(*%%%%%%%%%%%%%% Call Robots to Tool and Give Them, Task ID, Fixture ID and Model ID %%%%%%%%%%%%%%%%%*)
	(* Perform Call To Tool*)
	Tool_Call_ForLoadRobots1:= Enable_Motion AND (NOT Cell_In_Services OR NOT Load_Robots_Clear1)
						AND Start_Load_Robots1 AND NOT Start_Load_Robots2 AND NOT Start_Weld_Robots AND NOT Start_Seal_Robots AND NOT Start_Stud_Robots
						AND NOT Start_Unload_Robots1 AND NOT Start_Unload_Robots2 AND NOT Start_TurntableA AND NOT Start_TurntableB;
	Tool_Call_ForLoadRobots2:= Enable_Motion AND (NOT Cell_In_Services OR NOT Load_Robots_Clear2)
						AND NOT Start_Load_Robots1 AND Start_Load_Robots2 AND NOT Start_Weld_Robots AND NOT Start_Seal_Robots AND NOT Start_Stud_Robots
						AND NOT Start_Unload_Robots1 AND NOT Start_Unload_Robots2 AND NOT Start_TurntableA AND NOT Start_TurntableB;
	Tool_Call_ForSealRobots:=Enable_Motion AND (NOT Cell_In_Services OR NOT Seal_Robots_Clear)
						AND NOT Start_Load_Robots1 AND NOT Start_Load_Robots2 AND NOT Start_Weld_Robots AND Start_Seal_Robots AND NOT Start_Stud_Robots
						AND NOT Start_Unload_Robots1 AND NOT Start_Unload_Robots2 AND NOT Start_TurntableA AND NOT Start_TurntableB;
	Tool_Call_ForStudRobots:=Enable_Motion AND (NOT Cell_In_Services OR NOT Stud_Robots_Clear)
						AND NOT Start_Load_Robots1 AND NOT Start_Load_Robots2 AND NOT Start_Weld_Robots AND NOT Start_Seal_Robots AND Start_Stud_Robots
						AND NOT Start_Unload_Robots1 AND NOT Start_Unload_Robots2 AND NOT Start_TurntableA AND NOT Start_TurntableB;
	Tool_Call_ForSweepA:= Enable_Motion AND (NOT Cell_In_Services OR NOT TurntableA_Clear)
						AND NOT Start_Load_Robots1 AND NOT Start_Load_Robots2 AND NOT Start_Weld_Robots AND NOT Start_Seal_Robots AND NOT Start_Stud_Robots
						AND NOT Start_Unload_Robots1 AND NOT Start_Unload_Robots2 AND Start_TurntableA AND NOT Start_TurntableB;
	Tool_Call_ForSweepB:= Enable_Motion AND (NOT Cell_In_Services OR NOT TurntableB_Clear)
						AND NOT Start_Load_Robots1 AND NOT Start_Load_Robots2 AND NOT Start_Weld_Robots AND NOT Start_Seal_Robots AND NOT Start_Stud_Robots
						AND NOT Start_Unload_Robots1 AND NOT Start_Unload_Robots2 AND NOT Start_TurntableA AND Start_TurntableB;
	Tool_Call_ForWeldRobots:= Enable_Motion AND (NOT Cell_In_Services OR NOT Weld_Robots_Clear)
						AND NOT Start_Load_Robots1 AND NOT Start_Load_Robots2 AND Start_Weld_Robots AND NOT Start_Seal_Robots AND NOT Start_Stud_Robots
						AND NOT Start_Unload_Robots1 AND NOT Start_Unload_Robots2 AND NOT Start_TurntableA AND NOT Start_TurntableB;
	Tool_Call_ForUnloadRobots1:= Enable_Motion AND (NOT Cell_In_Services OR NOT Unload_Robots_Clear1)
						AND NOT Start_Load_Robots1 AND NOT Start_Load_Robots2 AND NOT Start_Weld_Robots AND NOT Start_Seal_Robots AND NOT Start_Stud_Robots
						AND Start_Unload_Robots1 AND NOT Start_Unload_Robots2 AND NOT Start_TurntableA AND NOT Start_TurntableB;
	Tool_Call_ForUnloadRobots2:= Enable_Motion AND (NOT Cell_In_Services OR NOT Unload_Robots_Clear2)
						AND NOT Start_Load_Robots1 AND NOT Start_Load_Robots2 AND NOT Start_Weld_Robots AND NOT Start_Seal_Robots AND NOT Start_Stud_Robots
						AND NOT Start_Unload_Robots1 AND Start_Unload_Robots2 AND NOT Start_TurntableA AND NOT Start_TurntableB;



	(*Allow Robots to Proceed Into Tool*)
	(*!!!!!This is the final OK to allow Robots Into the Tool Area, So it Better Be Ready!!!!!!!*)
	IF Enable_Motion
		THEN
			IF Load_Robots_Proceed1 AND Load_Robots_WorkingOK1 AND Load_Robots_Clear2 AND Seal_Robots_Clear AND Stud_Robots_Clear AND Turntable_Clear AND Weld_Robots_Clear AND Unload_Robots_Clear
				THEN Robots_Clear_ToProceed:=TRUE;
			ELSIF Load_Robots_Proceed2 AND Load_Robots_WorkingOK2 AND Load_Robots_Clear1 AND Seal_Robots_Clear AND Stud_Robots_Clear AND Turntable_Clear AND Weld_Robots_Clear AND Unload_Robots_Clear
				THEN Robots_Clear_ToProceed:=TRUE;
			ELSIF Seal_Robots_Proceed AND Seal_Robots_WorkingOK AND Load_Robots_Clear AND Stud_Robots_Clear AND Turntable_Clear AND Weld_Robots_Clear AND Unload_Robots_Clear
				THEN Robots_Clear_ToProceed:=TRUE;
			ELSIF Stud_Robots_Proceed AND Stud_Robots_WorkingOK AND Load_Robots_Clear AND Seal_Robots_Clear AND Turntable_Clear AND Weld_Robots_Clear AND Unload_Robots_Clear
				THEN Robots_Clear_ToProceed:=TRUE;
			ELSIF Weld_Robots_Proceed AND Weld_Robots_WorkingOK AND Load_Robots_Clear AND Seal_Robots_Clear AND Stud_Robots_Clear AND Turntable_Clear AND Unload_Robots_Clear
				THEN Robots_Clear_ToProceed:=TRUE;
			ELSIF Unload_Robots_Proceed1 AND Unload_Robots_WorkingOK1 AND Load_Robots_Clear AND Seal_Robots_Clear AND Stud_Robots_Clear AND Turntable_Clear AND Weld_Robots_Clear AND Unload_Robots_Clear2
				THEN Robots_Clear_ToProceed:=TRUE;
			ELSIF Unload_Robots_Proceed2 AND Unload_Robots_WorkingOK2 AND Load_Robots_Clear AND Seal_Robots_Clear AND Stud_Robots_Clear AND Turntable_Clear AND Weld_Robots_Clear AND Unload_Robots_Clear1
				THEN Robots_Clear_ToProceed:=TRUE;
			ELSE Robots_Clear_ToProceed:= FALSE;
			END_IF;
		ELSE Robots_Clear_ToProceed:= FALSE;
	END_IF;

(*+++++++++++++++++++++++++++++++++++++++++++++++ Task Complete Acks ++++++++++++++++++++++++++*)
	(*1st Load Complete Ack*)
	Load_Complete1_Ack:= Load_Robots_Complete1 AND Load_Complete1;

	(*2nd Load Complete Ack*)
	Load_Complete2_Ack:= Load_Robots_Complete2 AND Load_Complete2;

	(*Seal Complete Ack*)
	Seal_Complete_Ack:= Seal_Robots_Complete AND Sealing_Complete;

	(*Stud Complete Ack*)
	Stud_Complete_Ack:= Stud_Robots_Complete AND Stud_Complete;

	(*Sweep Complete ACK*)
	TurnA_Complete_Ack := TurntableA_Complete AND TurntableA_At_Robot;
	TurnB_Complete_Ack := TurntableB_Complete AND TurntableB_At_Robot;

	(*Weld Complete Ack*)
	Weld_Complete_Ack:= Weld_Robots_Complete AND Welding_Complete;

	(*Unload Complete Ack*)
	Unload_Complete1_Ack:= Unload_Robots_Complete1 AND Unload_Complete;

	(*Unload Complete Ack*)
	Unload_Complete2_Ack:= Unload_Robots_Complete2 AND Unload_Complete;















(*end*)
END_ACTION

ACTION Status_and_Faults:



(*^^^^^^^^^^^^^^^^^^^^^^^^^^^^^^^^^^^^^^ General Visualization ^^^^^^^^^^^^^^^^^^^^^^^^^^^^^^^^^^^^*)
	(*For Ready to Load Indicators*)
		(*Flash when tool should be loaded but load is not complete*)
		IF In_Auto AND Tool_At_Home AND NOT Welding_Complete AND All_Robots_Clear AND NOT All_Sensors_On.2
			THEN
				Ready_To_Load:= Pulse_500mS;
				(*Go solid when tool has been loaded properly*)
				(*Go solid when tool is ready to be unloaded*)
		ELSIF In_Auto AND All_Robots_Clear  AND ((Tool_At_Home AND NOT Welding_Complete AND All_Sensors_On.2 AND NOT Enable_Motion)
			OR (Tool_At_Unload.0 AND Welding_Complete AND (Sealing_Complete OR Sealer_Bypass) AND (Stud_Complete OR Stud_Bypass) AND TurntableA_At_Robot AND NOT All_Sensors_Off))
			THEN
				Ready_To_Load:= TRUE;
		ELSE
				Ready_To_Load:= FALSE;
		END_IF;
	(*For Red Stack Light Indicators*)
		Red_Lamp_Req:= PPFaults<>0 OR CLFaulted.0 OR CLFaulted.4 OR (NOT Sealer_Bypass AND MAIN.SL01.Disp1_Volume_NotOK AND (MAIN.R1.Task_ID_Ack=Seal_Fix01)) OR Load_Seq01.Faulted;


	(*Status Banners*)
		(*1 - Check Parts On Sub Check*)
		IF In_Auto AND NOT In_Manual AND NOT Cycle_Complete AND Tool_At_Load.4
			AND NOT Start_Load_Robots1 AND NOT Start_Load_Robots2 AND NOT Start_Seal_Robots AND NOT Start_Stud_Robots AND NOT Start_TurntableA
			AND NOT Start_TurntableB AND NOT Start_Weld_Robots AND NOT Start_Unload_Robots1 AND NOT Start_Unload_Robots2
			THEN
				IF NOT Dry_Cycle AND NOT All_Sensors_On.0
					THEN Status:= 1;
				ELSIF Dry_Cycle AND NOT Load_Complete1
					THEN Status:=1;
				END_IF;
		END_IF;
		(*2 - Sub Check OK*)
		IF In_Auto AND NOT In_Manual AND NOT Cycle_Complete AND Tool_At_Load.5
			AND NOT Start_Load_Robots1 AND NOT Start_Load_Robots2 AND NOT Start_Seal_Robots AND NOT Start_Stud_Robots AND NOT Start_TurntableA
			AND NOT Start_TurntableB AND NOT Start_Weld_Robots AND NOT Start_Unload_Robots1 AND NOT Start_Unload_Robots2
			THEN
				IF NOT Dry_Cycle AND NOT All_Sensors_On.1
					THEN Status:= 2;
				ELSIF Dry_Cycle AND NOT Load_Complete2
					THEN Status:=2;
				END_IF;
		END_IF;
		(*3 - Load Main Part*)
		IF In_Auto AND NOT In_Manual AND NOT Cycle_Complete AND Tool_At_Home
			AND NOT Start_Load_Robots1 AND NOT Start_Load_Robots2 AND NOT Start_Seal_Robots AND NOT Start_Stud_Robots AND NOT Start_TurntableA
			AND NOT Start_TurntableB AND NOT Start_Weld_Robots AND NOT Start_Unload_Robots1 AND NOT Start_Unload_Robots2
			THEN
				IF NOT Dry_Cycle AND NOT All_Sensors_On.2
					THEN Status:= 3;
				ELSIF Dry_Cycle AND NOT Load_Complete
					THEN Status:=3;
				END_IF;
		END_IF;
		(*10 - Load Parts Onto Tool*)
		IF In_Auto AND NOT In_Manual AND NOT Cycle_Complete AND Tool_At_Load.0
			AND NOT Start_Load_Robots1 AND NOT Start_Load_Robots2 AND NOT Start_Seal_Robots AND NOT Start_Stud_Robots AND NOT Start_TurntableA
			AND NOT Start_TurntableB AND NOT Start_Weld_Robots AND NOT Start_Unload_Robots1 AND NOT Start_Unload_Robots2
			THEN
				IF NOT Dry_Cycle AND NOT All_Sensors_On.2
					THEN Status:= 10;
				ELSIF Dry_Cycle AND NOT Load_Complete
					THEN Status:=10;
				END_IF;
		END_IF;
		(*11 - Robot(s) Loading*)
		IF ((Start_Load_Robots1 OR  Load_Robots_WorkingOK1) OR (Start_Load_Robots2 OR  Load_Robots_WorkingOK2)) AND In_Auto AND NOT In_Manual
			AND NOT Start_Seal_Robots AND NOT Start_Stud_Robots AND NOT Start_TurntableA
			AND NOT Start_TurntableB AND NOT Start_Weld_Robots AND NOT Start_Unload_Robots1 AND NOT Start_Unload_Robots2
			THEN Status:= 11;
		END_IF;
		(*12 - Parts Loaded OK*)
		IF In_Auto AND NOT In_Manual AND NOT Cycle_Complete
			AND NOT Start_Load_Robots1 AND NOT Start_Load_Robots2 AND NOT Start_Seal_Robots AND NOT Start_Stud_Robots AND NOT Start_TurntableA
			 AND NOT Start_TurntableB AND NOT Start_Weld_Robots AND NOT Start_Unload_Robots1 AND NOT Start_Unload_Robots2
			THEN
				IF (All_Sensors_On.2 AND Tool_At_Load.1) AND NOT Dry_Cycle
					THEN Status:= 12;
				ELSIF Load_Complete
					THEN Status:= 12;
				END_IF;
		END_IF;
		(*19 - Robot(s) Stud*)
		IF (Start_Stud_Robots OR Stud_Robots_WorkingOK) AND In_Auto AND NOT In_Manual
			AND NOT Start_Load_Robots1 AND NOT Start_Load_Robots2 AND NOT Start_Weld_Robots AND NOT Start_Seal_Robots AND NOT Start_TurntableA
			 AND NOT Start_TurntableB AND NOT Start_Unload_Robots1 AND NOT Start_Unload_Robots2
			THEN Status:= 19;
		END_IF;
		(*20 - Robot(s) Sealing*)
		IF (Start_Seal_Robots OR Seal_Robots_WorkingOK) AND In_Auto AND NOT In_Manual
			AND NOT Start_Load_Robots1 AND NOT Start_Load_Robots2 AND NOT Start_Weld_Robots AND NOT Start_Stud_Robots AND NOT Start_TurntableA
			 AND NOT Start_TurntableB AND NOT Start_Unload_Robots1 AND NOT Start_Unload_Robots2
			THEN Status:= 20;
		END_IF;
		(*21 - Robot(s) Welding*)
		IF (Start_Weld_Robots OR Weld_Robots_WorkingOK) AND In_Auto AND NOT In_Manual
			AND NOT Start_Load_Robots1 AND NOT Start_Load_Robots2 AND NOT Start_Seal_Robots AND NOT Start_Stud_Robots AND NOT Start_TurntableA
			 AND NOT Start_TurntableB AND NOT Start_Unload_Robots1 AND NOT Start_Unload_Robots2
			THEN Status:= 21;
		END_IF;
		(*22 - Welding Complete / Ready for Unload*)
		IF In_Auto AND NOT In_Manual AND NOT Cycle_Complete AND Welding_Complete AND (Sub1_Weld_Complete OR Sub2_Weld_Complete OR Sub3_Weld_Complete OR Sub4_Weld_Complete OR Sub5_Weld_Complete)
			AND NOT Start_Load_Robots1 AND NOT Start_Load_Robots2 AND NOT Start_Seal_Robots AND NOT Start_Stud_Robots AND NOT Start_TurntableA
			AND NOT Start_TurntableB AND NOT Start_Weld_Robots AND NOT Start_Unload_Robots1 AND NOT Start_Unload_Robots2 AND TurntableA_At_Robot
			THEN Status:= 22;
		END_IF;
		(*26 - Ready for Rotate*)
		IF (Start_TurntableA OR Start_TurntableB) AND In_Auto AND NOT In_Manual
			AND NOT Start_Load_Robots1 AND NOT Start_Load_Robots2 AND NOT Start_Seal_Robots AND NOT Start_Stud_Robots
			AND NOT Start_Weld_Robots AND NOT Start_Unload_Robots1 AND NOT Start_Unload_Robots2
			THEN Status := 26;
		END_IF;
		(*31 - Robot(s) Unloading*)
		IF (Start_Unload_Robots1 OR Unload_Robots_WorkingOK1 OR Start_Unload_Robots2 OR Unload_Robots_WorkingOK2) AND In_Auto AND NOT In_Manual
			AND NOT Start_Load_Robots1 AND NOT Start_Load_Robots2 AND NOT Start_Seal_Robots AND NOT Start_Stud_Robots AND NOT Start_TurntableA
			AND NOT Start_TurntableB AND NOT Start_Weld_Robots
			THEN Status:= 31;
		END_IF;
		(*32 - Unload Complete*)
		IF In_Auto AND NOT In_Manual AND NOT Cycle_Complete AND Unload_Complete AND All_Sensors_Off
			AND NOT Start_Load_Robots1 AND NOT Start_Load_Robots2 AND NOT Start_Seal_Robots AND NOT Start_Stud_Robots AND NOT Start_TurntableA
			AND NOT Start_TurntableB AND NOT Start_Weld_Robots AND NOT Start_Unload_Robots1 AND NOT Start_Unload_Robots2
			THEN Status:= 32;
		END_IF;
		(*42 - Cycle Complete*)
		IF In_Auto AND NOT In_Manual AND Cycle_Complete AND All_Sensors_Off
			THEN Status:= 42;
		END_IF;
		(*50 - In Manual*)
		IF In_Manual
			THEN Status:= 50;
		END_IF;
		(*51 - Clamp Fault*)
		IF (CLFaults1>0 OR CLFaults2>0 OR CLFaults3>0 OR CLFaults4>0) AND In_Auto AND NOT In_Manual
			THEN Status:= 51;
		END_IF;
		(*52 - Part Present Sensor Fault*)
		IF PPFaults>0 AND In_Auto AND NOT In_Manual
			THEN Status:= 52;
		END_IF;
		(*53 - Nut Checks Failed Call QA*)
		IF QAChecks_Failed AND In_Auto AND NOT In_Manual
			THEN Status:= 53;
		END_IF;
		(*54 - Sealer Failed Call QA*)
		IF NOT Sealer_Bypass AND (MAIN.SL01.Disp1_Volume_NotOK AND (MAIN.R1.Task_ID_Ack=Seal_Fix01)) AND In_Auto AND NOT In_Manual
			THEN Status:= 54;
		END_IF;
		(*55 - Load Sequence Fault Call QA*)
		IF Load_Seq01.Faulted AND In_Auto AND NOT In_Manual
			THEN Status:= 55;
		END_IF;



(*$$$$$$$$$$$$$$$$$$$$$$$$$$$$$$$$$$$$$$$$$$$$$$$$$$$ Faults $$$$$$$$$$$$$$$$$$$$$$$$$$$$$$$$$$$$$$$$$$$$$$$$$$$$$$$*)

	(*Clamp/Cylider Faults Group 1*)
		IF CLFaults1>0
			THEN CLFaulted.1:=TRUE;
		ELSE
			CLFaulted.1:=FALSE;
		END_IF;
	(*Clamp/Cylider Faults Group 2*)
		IF CLFaults2>0
			THEN CLFaulted.2:=TRUE;
		ELSE
			CLFaulted.2:=FALSE;
		END_IF;
	(*Clamp/Cylider Faults Group 3*)
		IF CLFaults3>0
			THEN CLFaulted.3:=TRUE;
		ELSE
			CLFaulted.3:=FALSE;
		END_IF;
	(*Clamp/Cylinder Faults Group 4 - Reserved Flag for QA Check Motion Faults*)
		IF CLFaults4>0
			THEN CLFaulted.4:=TRUE;
		ELSE
			CLFaulted.4:=FALSE;
		END_IF;
	(*Bit 0 is designated as ANY Clamp Group Faulted*)
	IF CLFaulted.1 OR CLFaulted.2 OR CLFaulted.3
		THEN CLFaulted.0:= TRUE;
	ELSE CLFaulted.0 := FALSE;
	END_IF;

	(*Part Present Sensor Faults*)
		IF (PPFaults>0) OR (PPFaults1>0) OR (PPFaults2>0)
			THEN PPFaulted.0:=TRUE;
		ELSE
			PPFaulted.0:=FALSE;
		END_IF;
























(*end*)
END_ACTION

ACTION Task_Fix_Model_IDs:


	(*Develop Task IDs - See Global Variable, "TaskID_Record"*)

	IF (Start_Load_Robots1 OR Start_Load_Robots2) AND Enable_Motion
		THEN Task_ID:= Dropoff_Fix01;
	ELSIF Start_Seal_Robots AND Enable_Motion
		THEN Task_ID:= Seal_Fix01;
	ELSIF Start_Stud_Robots AND Enable_Motion
		THEN Task_ID:= Stud_Fix01;
	ELSIF Start_Weld_Robots AND Enable_Motion
		THEN Task_ID:= Weld_Fix01;
	ELSIF Start_TurnTableA AND Enable_Motion
		THEN Task_ID:= Sweep_Fix01;
	ELSIF (Start_Unload_Robots1 OR Start_Unload_Robots2) AND Enable_Motion
		THEN Task_ID:= Pickup_Fix01;
	ELSE Task_ID:= 0;
	END_IF;

	(*Develop Fixture ID*)
	Fix_ID:= N00.ID;					(*In Future Map Beckhoff Dip Switch Data From IP67 Block to Here*)

	(*Develop Model ID*)
	(*If there is no model, but running fix01, we need to set model for table sweep - then blanks modelID after*)
	IF All_Sensors_Off AND Turntable_Bypassed AND TurntableB_At_Robot
		THEN
		Model_ID:= 1;
		ELSE
		Model_ID:= Discrete_In.ModelData;
	END_IF
END_ACTION

ACTION Tool_States:


(*+++++++++++THIS AREA IS CUSTOM PER INSTALLATION AND WILL HAVE TO BE MODIFIED PER +++++++++++++*)
(*+++++++++++THIS AREA IS CUSTOM PER INSTALLATION AND WILL HAVE TO BE MODIFIED PER +++++++++++++*)


(*
						 MODEL ID MAP
					 -------------------
				Model ID :  Part ID  :   Tooling ID
					1  	 : 	 504     :     42
					2	 :   524     :	   42
					3	 :   543     :	   47
					4	 :   526     :	   46
					5	 :   536     :	   45
					6	 :   550     :	   44
					7	 :   571     :	   43
	
*)
	

	(*Tooling Position at Home*)
				Tool_At_HOME:= (((Model_ID=3) OR (Model_ID=10)) AND Clamp1RETD AND Clamp2RETD AND Clamp3RETD AND Clamp4RETD
							AND Clamp5RETD AND Clamp6RETD AND Clamp7RETD AND Clamp8RETD
							AND Clamp9RETD AND Clamp10RETD AND Clamp11RETD AND Clamp12RETD
							AND Clamp13RETD AND Clamp14RETD AND Clamp15RETD AND Clamp16RETD
							AND Clamp17RETD AND Clamp18RETD AND Clamp19RETD AND Clamp20RETD
							AND Clamp21RETD AND Clamp22RETD AND Clamp23RETD AND Clamp24RETD
							AND Clamp25RETD AND Clamp26RETD AND Clamp27RETD AND Clamp28RETD
							AND Clamp29RETD AND Clamp30RETD AND Clamp31RETD AND Clamp32RETD
							AND Clamp33RETD AND Clamp34RETD AND Clamp35RETD AND Clamp36RETD
							AND Clamp37RETD AND Clamp38RETD AND Pin1ADVD AND Pin2ADVD AND Pin3RETD 
							AND Pin4ADVD AND Pin5ADVD AND Pin6RETD AND Pin7ADVD AND Pin8ADVD
							AND Slide1ADVD AND Slide2ADVD AND Slide3RETD AND Slide4ADVD AND Slide5RETD AND Slide6ADVD
							AND Slide7RETD AND Slide8ADVD AND Slide9RETD AND Slide10RETD AND Slide11ADVD AND Slide12RETD
							AND Slide13RETD AND Slide14ADVD AND Slide15ADVD)
							OR
								(((Model_ID<>3) AND (Model_ID<>10)) AND Clamp1RETD AND Clamp2RETD AND Clamp3RETD AND Clamp4RETD
							AND Clamp5RETD AND Clamp6RETD AND Clamp7RETD AND Clamp8RETD
							AND Clamp9RETD AND Clamp10RETD AND Clamp11RETD AND Clamp12RETD
							AND Clamp13RETD AND Clamp14RETD AND Clamp15RETD AND Clamp16RETD
							AND Clamp17RETD AND Clamp18RETD AND Clamp19RETD AND Clamp20RETD
							AND Clamp21RETD AND Clamp22RETD AND Clamp23RETD AND Clamp24RETD
							AND Clamp25RETD AND Clamp26RETD AND Clamp27RETD AND Clamp28RETD
							AND Clamp29RETD AND Clamp30RETD AND Clamp31RETD AND Clamp32RETD
							AND Clamp33RETD AND Clamp34RETD AND Clamp35RETD AND Clamp36RETD
							AND Clamp37RETD AND Clamp38RETD AND Pin1ADVD AND Pin2RETD AND Pin3RETD 
							AND Pin4ADVD AND Pin5RETD AND Pin6RETD AND Pin7RETD AND Pin8ADVD
							AND Slide1ADVD AND Slide2ADVD AND Slide3RETD AND Slide4ADVD AND Slide5RETD AND Slide6ADVD
							AND Slide7RETD AND Slide8ADVD AND Slide9RETD AND Slide10RETD AND Slide11ADVD AND Slide12RETD
							AND Slide13RETD AND Slide14ADVD AND Slide15ADVD);		

						
	(*Tooling Position for Operator Load*)
	IF ((Model_ID=3) OR (Model_ID=10)) THEN
		
				Tool_At_Load.0:= Clamp1RETD AND Clamp2RETD AND Clamp3RETD AND Clamp4RETD
							AND Clamp5RETD AND Clamp6RETD AND Clamp7RETD AND Clamp8RETD
							AND Clamp9RETD AND Clamp10RETD AND Clamp11RETD AND Clamp12RETD
							AND Clamp13RETD AND Clamp14RETD AND Clamp15RETD AND Clamp16RETD
							AND Clamp17RETD AND Clamp18RETD AND Clamp19RETD AND Clamp20RETD
							AND Clamp21RETD AND Clamp22RETD AND Clamp23RETD AND Clamp24RETD
							AND Clamp25RETD AND Clamp26RETD AND Clamp27RETD AND Clamp28RETD
							AND Clamp29RETD AND Clamp30RETD AND Clamp31RETD AND Clamp32RETD
							AND Clamp33RETD AND Clamp34RETD AND Clamp35RETD AND Clamp36RETD
							AND Clamp37RETD AND Clamp38RETD AND Pin1ADVD AND Pin2ADVD AND Pin3RETD 
							AND Pin4ADVD AND Pin5ADVD AND Pin6RETD AND Pin7ADVD AND Pin8ADVD
							AND Slide1ADVD AND Slide2ADVD AND Slide3RETD AND Slide4ADVD AND Slide5RETD AND Slide6ADVD
							AND Slide7RETD AND Slide8ADVD AND Slide9RETD AND Slide10RETD AND Slide11ADVD AND Slide12RETD
							AND Slide13RETD AND Slide14ADVD AND Slide15ADVD;
		ELSE
			
				Tool_At_Load.0:= Clamp1RETD AND Clamp2RETD AND Clamp3RETD AND Clamp4RETD
							AND Clamp5RETD AND Clamp6RETD AND Clamp7RETD AND Clamp8RETD
							AND Clamp9RETD AND Clamp10RETD AND Clamp11RETD AND Clamp12RETD
							AND Clamp13RETD AND Clamp14RETD AND Clamp15RETD AND Clamp16RETD
							AND Clamp17RETD AND Clamp18RETD AND Clamp19RETD AND Clamp20RETD
							AND Clamp21RETD AND Clamp22RETD AND Clamp23RETD AND Clamp24RETD
							AND Clamp25RETD AND Clamp26RETD AND Clamp27RETD AND Clamp28RETD
							AND Clamp29RETD AND Clamp30RETD AND Clamp31RETD AND Clamp32RETD
							AND Clamp33RETD AND Clamp34RETD AND Clamp35RETD AND Clamp36RETD
							AND Clamp37RETD AND Clamp38RETD AND Pin1ADVD AND Pin2RETD AND Pin3RETD 
							AND Pin4ADVD AND Pin5RETD AND Pin6RETD AND Pin7RETD AND Pin8ADVD
							AND Slide1ADVD AND Slide2ADVD AND Slide3RETD AND Slide4ADVD AND Slide5RETD AND Slide6ADVD
							AND Slide7RETD AND Slide8ADVD AND Slide9RETD AND Slide10RETD AND Slide11ADVD AND Slide12RETD
							AND Slide13RETD AND Slide14ADVD AND Slide15ADVD;
							
	END_IF		
	
	(*Tooling Position at Load Complete*)
	IF ((Model_ID =1) OR (Model_ID=8) OR (Model_ID =2) OR (Model_ID=9)) THEN
		
				Tool_At_Load.1:= (Clamp1ADVD AND Clamp2ADVD AND Clamp3ADVD AND Clamp4ADVD AND Clamp5ADVD
							AND Clamp6ADVD AND Clamp7ADVD AND Clamp8RETD AND Clamp9ADVD AND Clamp10RETD
							AND Clamp11ADVD AND Clamp12ADVD AND Clamp13ADVD AND Clamp14ADVD AND Clamp15ADVD
							AND Clamp16ADVD AND Clamp17ADVD AND Clamp18ADVD AND Clamp19ADVD AND Clamp20ADVD
							AND Clamp21ADVD AND Clamp22ADVD AND Clamp23RETD AND Clamp24RETD AND Clamp25RETD
							AND Clamp26ADVD AND Clamp27RETD AND Clamp28ADVD AND Clamp29ADVD AND Clamp30ADVD
							AND Clamp31RETD AND Clamp32ADVD AND Clamp33ADVD AND Clamp34ADVD AND Clamp35ADVD
							AND Clamp36ADVD AND Clamp37ADVD AND Clamp38ADVD AND Pin1ADVD AND Pin2RETD
							AND Pin3RETD AND Pin4ADVD AND Pin5RETD AND Pin6RETD AND Pin7RETD AND Pin8ADVD
							AND Slide1ADVD AND Slide2ADVD AND Slide3ADVD AND Slide4ADVD AND Slide5ADVD
							AND Slide6ADVD AND Slide7ADVD AND Slide8ADVD AND Slide9ADVD AND Slide10ADVD
							AND Slide11ADVD AND Slide12ADVD AND Slide13ADVD AND Slide14ADVD AND Slide15ADVD)
							OR (*After Hand Clamps*)
							(Clamp1RETD AND Clamp2RETD AND Clamp3RETD AND Clamp4RETD AND Clamp5RETD
							AND Clamp6ADVD AND Clamp7RETD AND Clamp8RETD AND Clamp9ADVD AND Clamp10RETD
							AND Clamp11RETD AND Clamp12RETD AND Clamp13RETD AND Clamp14RETD AND Clamp15RETD
							AND Clamp16RETD AND Clamp17RETD AND Clamp18RETD AND Clamp19RETD AND Clamp20RETD
							AND Clamp21ADVD AND Clamp22RETD AND Clamp23RETD AND Clamp24RETD AND Clamp25RETD
							AND Clamp26RETD AND Clamp27RETD AND Clamp28RETD AND Clamp29RETD AND Clamp30ADVD
							AND Clamp31RETD AND Clamp32RETD AND Clamp33RETD AND Clamp34RETD AND Clamp35RETD
							AND Clamp36ADVD AND Clamp37RETD AND Clamp38RETD AND Pin1ADVD AND Pin2RETD
							AND Pin3RETD AND Pin4ADVD AND Pin5RETD AND Pin6RETD AND Pin7RETD AND Pin8ADVD
							AND Slide1ADVD AND Slide2ADVD AND Slide3RETD AND Slide4ADVD AND Slide5RETD
							AND Slide6ADVD AND Slide7RETD AND Slide8ADVD AND Slide9RETD AND Slide10RETD
							AND Slide11ADVD AND Slide12RETD AND Slide13RETD AND Slide14ADVD AND Slide15ADVD);
							
		ELSIF ((Model_ID=3) OR (Model_ID=10)) THEN
			
				Tool_At_Load.1:= Clamp1ADVD AND Clamp2ADVD AND Clamp3ADVD AND Clamp4ADVD AND Clamp5ADVD
							AND Clamp6ADVD AND Clamp7RETD AND Clamp8ADVD AND Clamp9ADVD AND Clamp10ADVD
							AND Clamp11ADVD AND Clamp12ADVD AND Clamp13ADVD AND Clamp14ADVD AND Clamp15ADVD
							AND Clamp16ADVD AND Clamp17ADVD AND Clamp18ADVD AND Clamp19ADVD AND Clamp20ADVD
							AND Clamp21ADVD AND Clamp22RETD AND Clamp23RETD AND Clamp24ADVD AND Clamp25RETD
							AND Clamp26RETD AND Clamp27ADVD AND Clamp28ADVD AND Clamp29ADVD AND Clamp30ADVD
							AND Clamp31ADVD AND Clamp32ADVD AND Clamp33ADVD AND Clamp34ADVD AND Clamp35RETD
							AND Clamp36ADVD AND Clamp37ADVD AND Clamp38ADVD AND Pin1ADVD AND Pin2ADVD
							AND Pin3ADVD AND Pin4ADVD AND Pin5ADVD AND Pin6ADVD AND Pin7ADVD AND Pin8ADVD
							AND Slide1ADVD AND Slide2ADVD AND Slide3ADVD AND Slide4ADVD AND Slide5ADVD
							AND Slide6ADVD AND Slide7ADVD AND Slide8ADVD AND Slide9ADVD AND Slide10ADVD
							AND Slide11ADVD AND Slide12ADVD AND Slide13ADVD AND Slide14ADVD AND Slide15ADVD
							OR (*After Hand Clamps*)
							(Clamp1RETD AND Clamp2RETD AND Clamp3RETD AND Clamp4RETD AND Clamp5RETD
							AND Clamp6ADVD AND Clamp7RETD AND Clamp8ADVD AND Clamp9ADVD AND Clamp10ADVD
							AND Clamp11RETD AND Clamp12RETD AND Clamp13RETD AND Clamp14RETD AND Clamp15RETD
							AND Clamp16RETD AND Clamp17RETD AND Clamp18RETD AND Clamp19RETD AND Clamp20RETD
							AND Clamp21ADVD AND Clamp22RETD AND Clamp23RETD AND Clamp24ADVD AND Clamp25RETD
							AND Clamp26RETD AND Clamp27ADVD AND Clamp28RETD AND Clamp29RETD AND Clamp30ADVD
							AND Clamp31ADVD AND Clamp32RETD AND Clamp33RETD AND Clamp34RETD AND Clamp35RETD
							AND Clamp36ADVD AND Clamp37RETD AND Clamp38RETD AND Pin1ADVD AND Pin2ADVD
							AND Pin3RETD AND Pin4ADVD AND Pin5ADVD AND Pin6RETD AND Pin7ADVD AND Pin8ADVD
							AND Slide1ADVD AND Slide2ADVD AND Slide3RETD AND Slide4ADVD AND Slide5RETD
							AND Slide6ADVD AND Slide7RETD AND Slide8ADVD AND Slide9RETD AND Slide10RETD
							AND Slide11ADVD AND Slide12RETD AND Slide13RETD AND Slide14ADVD AND Slide15ADVD);
							
		ELSIF 			   (Model_ID=4) OR (Model_ID=5) OR (Model_ID=6) OR (Model_ID=7)
						OR (Model_ID=11) OR (Model_ID=12) OR (Model_ID=13) OR (Model_ID=14)
						OR (Model_ID=15) OR (Model_ID=16) OR (Model_ID=17) OR (Model_ID=18)
						OR (Model_ID=19) OR (Model_ID=20) OR (Model_ID=21) OR (Model_ID=22) THEN
			
				Tool_At_Load.1:= (Clamp1ADVD AND Clamp2ADVD AND Clamp3ADVD AND Clamp4ADVD AND Clamp5ADVD
							AND Clamp6ADVD AND Clamp7ADVD AND Clamp8RETD AND Clamp9ADVD AND Clamp10RETD
							AND Clamp11ADVD AND Clamp12ADVD AND Clamp13ADVD AND Clamp14ADVD AND Clamp15ADVD
							AND Clamp16ADVD AND Clamp17ADVD AND Clamp18ADVD AND Clamp19ADVD AND Clamp20ADVD
							AND Clamp21ADVD AND Clamp22RETD AND Clamp23ADVD AND Clamp24RETD AND Clamp25ADVD
							AND Clamp26RETD AND Clamp27RETD AND Clamp28ADVD AND Clamp29ADVD AND Clamp30ADVD
							AND Clamp31RETD AND Clamp32ADVD AND Clamp33ADVD AND Clamp34ADVD AND Clamp35ADVD
							AND Clamp36ADVD AND Clamp37ADVD AND Clamp38ADVD AND Pin1ADVD AND Pin2RETD
							AND Pin3RETD AND Pin4ADVD AND Pin5RETD AND Pin6RETD AND Pin7RETD AND Pin8ADVD
							AND Slide1ADVD AND Slide2ADVD AND Slide3ADVD AND Slide4ADVD AND Slide5ADVD
							AND Slide6ADVD AND Slide7ADVD AND Slide8ADVD AND Slide9ADVD AND Slide10ADVD
							AND Slide11ADVD AND Slide12ADVD AND Slide13ADVD AND Slide14ADVD AND Slide15ADVD)
							OR (*After Hand Clamps*)
							(Clamp1RETD AND Clamp2RETD AND Clamp3RETD AND Clamp4RETD AND Clamp5RETD
							AND Clamp6ADVD AND Clamp7RETD AND Clamp8RETD AND Clamp9ADVD AND Clamp10RETD
							AND Clamp11RETD AND Clamp12RETD AND Clamp13RETD AND Clamp14RETD AND Clamp15RETD
							AND Clamp16RETD AND Clamp17RETD AND Clamp18RETD AND Clamp19RETD AND Clamp20RETD
							AND Clamp21ADVD AND Clamp22RETD AND Clamp23RETD AND Clamp24RETD AND Clamp25RETD
							AND Clamp26RETD AND Clamp27RETD AND Clamp28RETD AND Clamp29RETD AND Clamp30ADVD
							AND Clamp31RETD AND Clamp32RETD AND Clamp33RETD AND Clamp34RETD AND Clamp35RETD
							AND Clamp36ADVD AND Clamp37RETD AND Clamp38RETD AND Pin1ADVD AND Pin2RETD
							AND Pin3RETD AND Pin4ADVD AND Pin5RETD AND Pin6RETD AND Pin7RETD AND Pin8ADVD
							AND Slide1ADVD AND Slide2ADVD AND Slide3RETD AND Slide4ADVD AND Slide5RETD
							AND Slide6ADVD AND Slide7RETD AND Slide8ADVD AND Slide9RETD AND Slide10ADVD
							AND Slide11ADVD AND Slide12RETD AND Slide13RETD AND Slide14ADVD AND Slide15ADVD);
							
	END_IF
	

(*Unused tool state - for reference BdB*)
	Tool_At_Load.2:= ((Model_ID=4) //526
							AND Clamp1ADVD AND Clamp2ADVD AND Clamp3ADVD AND Clamp4ADVD AND Clamp5ADVD
							AND Clamp6ADVD AND Clamp7ADVD AND Clamp8RETD AND Clamp9ADVD AND Clamp10RETD
							AND Clamp11ADVD AND Clamp12ADVD AND Clamp13ADVD AND Clamp14ADVD AND Clamp15ADVD
							AND Clamp16ADVD AND Clamp17ADVD AND Clamp18ADVD AND Clamp19ADVD AND Clamp20ADVD
							AND Clamp21ADVD AND Clamp22RETD AND Clamp23ADVD AND Clamp24RETD AND Clamp25ADVD
							AND Clamp26RETD AND Clamp27RETD AND Clamp28ADVD AND Clamp29ADVD AND Clamp30ADVD
							AND Clamp31RETD AND Clamp32ADVD AND Clamp33ADVD AND Clamp34ADVD AND Clamp35ADVD
							AND Clamp36ADVD AND Clamp37ADVD AND Clamp38ADVD AND Pin1ADVD AND Pin2RETD
							AND Pin3RETD AND Pin4ADVD AND Pin5RETD AND Pin6RETD AND Pin7RETD AND Pin8ADVD
							AND Slide1ADVD AND Slide2ADVD (*AND Slide3ADVD*, tooling issues*) AND Slide4ADVD AND Slide5ADVD
							AND Slide6ADVD AND Slide7RETD (*AND Slide7ADVD, wrong way around*) AND Slide8ADVD AND Slide9ADVD AND Slide10ADVD
							AND Slide11ADVD (*AND Slide12ADVD AND Slide13ADVD* tooling issues*) AND Slide14ADVD AND Slide15ADVD);
	Tool_At_Load.3:= FALSE;
	Tool_At_Load.4:= FALSE;


	Tool_At_Seal.0:= FALSE;
	Tool_At_Seal.1:= FALSE;
	Tool_At_Seal.2:= FALSE;
	Tool_At_Seal.3:= FALSE;
	Tool_At_Seal.4:= FALSE;


	Tool_At_Stud.0:= FALSE;
	Tool_At_Stud.1:= FALSE;
	Tool_At_Stud.2:= FALSE;
	Tool_At_Stud.3:= FALSE;
	Tool_At_Stud.4:= FALSE;


	IF ((Model_ID =1) OR (Model_ID=8) OR (Model_ID =2) OR (Model_ID=9)) THEN
		
				Tool_At_Rotate.0:= Clamp1ADVD AND Clamp2ADVD AND Clamp3ADVD AND Clamp4ADVD AND Clamp5ADVD
							AND Clamp6ADVD AND Clamp7ADVD AND Clamp8RETD AND Clamp9ADVD AND Clamp10RETD
							AND Clamp11ADVD AND Clamp12ADVD AND Clamp13ADVD AND Clamp14ADVD AND Clamp15ADVD
							AND Clamp16ADVD AND Clamp17ADVD AND Clamp18ADVD AND Clamp19ADVD AND Clamp20ADVD
							AND Clamp21ADVD AND Clamp22ADVD AND Clamp23RETD AND Clamp24RETD AND Clamp25RETD
							AND Clamp26ADVD AND Clamp27RETD AND Clamp28ADVD AND Clamp29ADVD AND Clamp30ADVD
							AND Clamp31RETD AND Clamp32ADVD AND Clamp33ADVD AND Clamp34ADVD AND Clamp35ADVD
							AND Clamp36ADVD AND Clamp37ADVD AND Clamp38ADVD AND Pin1ADVD AND Pin2RETD
							AND Pin3RETD AND Pin4ADVD AND Pin5RETD AND Pin6RETD AND Pin7RETD AND Pin8ADVD
							AND Slide1ADVD AND Slide2ADVD AND Slide3ADVD AND Slide4ADVD AND Slide5ADVD
							AND Slide6ADVD AND Slide7ADVD AND Slide8ADVD AND Slide9ADVD AND Slide10RETD
							AND Slide11ADVD AND Slide12ADVD AND Slide13ADVD AND Slide14ADVD AND Slide15ADVD;
							
		ELSIF ((Model_ID=3) OR (Model_ID=10)) THEN
			
				Tool_At_Rotate.0:= Clamp1ADVD AND Clamp2ADVD AND Clamp3ADVD AND Clamp4ADVD AND Clamp5ADVD
							AND Clamp6ADVD AND Clamp7RETD AND Clamp8ADVD AND Clamp9ADVD AND Clamp10ADVD
							AND Clamp11ADVD AND Clamp12ADVD AND Clamp13ADVD AND Clamp14ADVD AND Clamp15ADVD
							AND Clamp16ADVD AND Clamp17ADVD AND Clamp18ADVD AND Clamp19ADVD AND Clamp20ADVD
							AND Clamp21ADVD AND Clamp22RETD AND Clamp23RETD AND Clamp24ADVD AND Clamp25RETD
							AND Clamp26RETD AND Clamp27ADVD AND Clamp28ADVD AND Clamp29ADVD AND Clamp30ADVD
							AND Clamp31ADVD AND Clamp32ADVD AND Clamp33ADVD AND Clamp34ADVD AND Clamp35RETD
							AND Clamp36ADVD AND Clamp37ADVD AND Clamp38ADVD AND Pin1ADVD AND Pin2ADVD
							AND Pin3ADVD AND Pin4ADVD AND Pin5ADVD AND Pin6ADVD AND Pin7ADVD AND Pin8ADVD
							AND Slide1ADVD AND Slide2ADVD AND Slide3ADVD AND Slide4ADVD AND Slide5ADVD
							AND Slide6ADVD AND Slide7ADVD AND Slide8ADVD AND Slide9ADVD AND Slide10RETD
							AND Slide11ADVD AND Slide12ADVD AND Slide13ADVD AND Slide14ADVD AND Slide15ADVD;
							
		ELSIF 			   (Model_ID=4) OR (Model_ID=5) OR (Model_ID=6) OR (Model_ID=7)
						OR (Model_ID=11) OR (Model_ID=12) OR (Model_ID=13) OR (Model_ID=14)
						OR (Model_ID=15) OR (Model_ID=16) OR (Model_ID=17) OR (Model_ID=18)
						OR (Model_ID=19) OR (Model_ID=20) OR (Model_ID=21) OR (Model_ID=22) THEN
			
				Tool_At_Rotate.0:= Clamp1ADVD AND Clamp2ADVD AND Clamp3ADVD AND Clamp4ADVD AND Clamp5ADVD
							AND Clamp6ADVD AND Clamp7ADVD AND Clamp8RETD AND Clamp9ADVD AND Clamp10RETD
							AND Clamp11ADVD AND Clamp12ADVD AND Clamp13ADVD AND Clamp14ADVD AND Clamp15ADVD
							AND Clamp16ADVD AND Clamp17ADVD AND Clamp18ADVD AND Clamp19ADVD AND Clamp20ADVD
							AND Clamp21ADVD AND Clamp22RETD AND Clamp23ADVD AND Clamp24RETD AND Clamp25ADVD
							AND Clamp26RETD AND Clamp27RETD AND Clamp28ADVD AND Clamp29ADVD AND Clamp30ADVD
							AND Clamp31RETD AND Clamp32ADVD AND Clamp33ADVD AND Clamp34ADVD AND Clamp35ADVD
							AND Clamp36ADVD AND Clamp37ADVD AND Clamp38ADVD AND Pin1ADVD AND Pin2RETD
							AND Pin3RETD AND Pin4ADVD AND Pin5RETD AND Pin6RETD AND Pin7RETD AND Pin8ADVD
							AND Slide1ADVD AND Slide2ADVD AND Slide3ADVD AND Slide4ADVD AND Slide5ADVD
							AND Slide6ADVD AND Slide7ADVD AND Slide8ADVD AND Slide9ADVD AND Slide10ADVD
							AND Slide11ADVD AND Slide12ADVD AND Slide13ADVD AND Slide14ADVD AND Slide15ADVD;
	END_IF
				
	Tool_At_Rotate.1:= Clamp1RETD AND Clamp2RETD AND Clamp3RETD AND Clamp4RETD
							AND Clamp5RETD AND Clamp6RETD AND Clamp7RETD AND Clamp8RETD
							AND Clamp9RETD AND Clamp10RETD AND Clamp11RETD AND Clamp12RETD
							AND Clamp13RETD AND Clamp14RETD AND Clamp15RETD AND Clamp16RETD
							AND Clamp17RETD AND Clamp18RETD AND Clamp19RETD AND Clamp20RETD
							AND Clamp21RETD AND Clamp22RETD AND Clamp23RETD AND Clamp24RETD
							AND Clamp25RETD AND Clamp26RETD AND Clamp27RETD AND Clamp28RETD
							AND Clamp29RETD AND Clamp30RETD AND Clamp31RETD AND Clamp32RETD
							AND Clamp33RETD AND Clamp34RETD AND Clamp35RETD AND Clamp36RETD
							AND Clamp37RETD AND Clamp38RETD AND Pin1ADVD AND Pin2RETD AND Pin3RETD 
							AND Pin4ADVD AND Pin5RETD AND Pin6RETD AND Pin7RETD AND Pin8ADVD
							AND Slide1ADVD AND Slide2ADVD AND Slide3RETD AND Slide4ADVD AND Slide5RETD AND Slide6ADVD
							AND Slide7RETD AND Slide8ADVD AND Slide9RETD AND Slide10RETD AND Slide11ADVD AND Slide12RETD
							AND Slide13RETD AND Slide14ADVD AND Slide15ADVD;
	Tool_At_Rotate.2:= FALSE;
	Tool_At_Rotate.3:= FALSE;
	Tool_At_Rotate.4:= FALSE;


	IF ((Model_ID =1) OR (Model_ID=8) OR (Model_ID =2) OR (Model_ID=9)) THEN
		
				Tool_At_Weld.0:= Clamp1ADVD AND Clamp2ADVD AND Clamp3ADVD AND Clamp4ADVD AND Clamp5ADVD
							AND Clamp6ADVD AND Clamp7ADVD AND Clamp8RETD AND Clamp9ADVD AND Clamp10RETD
							AND Clamp11ADVD AND Clamp12ADVD AND Clamp13ADVD AND Clamp14ADVD AND Clamp15ADVD
							AND Clamp16ADVD AND Clamp17ADVD AND Clamp18ADVD AND Clamp19ADVD AND Clamp20ADVD
							AND Clamp21ADVD AND Clamp22ADVD AND Clamp23RETD AND Clamp24RETD AND Clamp25RETD
							AND Clamp26ADVD AND Clamp27RETD AND Clamp28ADVD AND Clamp29ADVD AND Clamp30ADVD
							AND Clamp31RETD AND Clamp32ADVD AND Clamp33ADVD AND Clamp34ADVD AND Clamp35ADVD
							AND Clamp36ADVD AND Clamp37ADVD AND Clamp38ADVD AND Pin1ADVD AND Pin2RETD
							AND Pin3RETD AND Pin4ADVD AND Pin5RETD AND Pin6RETD AND Pin7RETD AND Pin8ADVD
							AND Slide1ADVD AND Slide2ADVD AND Slide3ADVD AND Slide4ADVD AND Slide5ADVD
							AND Slide6ADVD AND Slide7ADVD AND Slide8ADVD AND Slide9ADVD AND Slide10RETD
							AND Slide11ADVD AND Slide12ADVD AND Slide13ADVD AND Slide14ADVD AND Slide15ADVD;
							
		ELSIF ((Model_ID=3) OR (Model_ID=10)) THEN
			
				Tool_At_Weld.0:= Clamp1ADVD AND Clamp2ADVD AND Clamp3ADVD AND Clamp4ADVD AND Clamp5ADVD
							AND Clamp6ADVD AND Clamp7RETD AND Clamp8ADVD AND Clamp9ADVD AND Clamp10ADVD
							AND Clamp11ADVD AND Clamp12ADVD AND Clamp13ADVD AND Clamp14ADVD AND Clamp15ADVD
							AND Clamp16ADVD AND Clamp17ADVD AND Clamp18ADVD AND Clamp19ADVD AND Clamp20ADVD
							AND Clamp21ADVD AND Clamp22RETD AND Clamp23RETD AND Clamp24ADVD AND Clamp25RETD
							AND Clamp26RETD AND Clamp27ADVD AND Clamp28ADVD AND Clamp29ADVD AND Clamp30ADVD
							AND Clamp31ADVD AND Clamp32ADVD AND Clamp33ADVD AND Clamp34ADVD AND Clamp35RETD
							AND Clamp36ADVD AND Clamp37ADVD AND Clamp38ADVD AND Pin1ADVD AND Pin2ADVD
							AND Pin3ADVD AND Pin4ADVD AND Pin5ADVD AND Pin6ADVD AND Pin7ADVD AND Pin8ADVD
							AND Slide1ADVD AND Slide2ADVD AND Slide3ADVD AND Slide4ADVD AND Slide5ADVD
							AND Slide6ADVD AND Slide7ADVD AND Slide8ADVD AND Slide9ADVD AND Slide10RETD
							AND Slide11ADVD AND Slide12ADVD AND Slide13ADVD AND Slide14ADVD AND Slide15ADVD;
							
		ELSIF 			   (Model_ID=4) OR (Model_ID=5) OR (Model_ID=6) OR (Model_ID=7)
						OR (Model_ID=11) OR (Model_ID=12) OR (Model_ID=13) OR (Model_ID=14)
						OR (Model_ID=15) OR (Model_ID=16) OR (Model_ID=17) OR (Model_ID=18)
						OR (Model_ID=19) OR (Model_ID=20) OR (Model_ID=21) OR (Model_ID=22) THEN
			
				Tool_At_Weld.0:= Clamp1ADVD AND Clamp2ADVD AND Clamp3ADVD AND Clamp4ADVD AND Clamp5ADVD
							AND Clamp6ADVD AND Clamp7ADVD AND Clamp8RETD AND Clamp9ADVD AND Clamp10RETD
							AND Clamp11ADVD AND Clamp12ADVD AND Clamp13ADVD AND Clamp14ADVD AND Clamp15ADVD
							AND Clamp16ADVD AND Clamp17ADVD AND Clamp18ADVD AND Clamp19ADVD AND Clamp20ADVD
							AND Clamp21ADVD AND Clamp22RETD AND Clamp23ADVD AND Clamp24RETD AND Clamp25ADVD
							AND Clamp26RETD AND Clamp27RETD AND Clamp28ADVD AND Clamp29ADVD AND Clamp30ADVD
							AND Clamp31RETD AND Clamp32ADVD AND Clamp33ADVD AND Clamp34ADVD AND Clamp35ADVD
							AND Clamp36ADVD AND Clamp37ADVD AND Clamp38ADVD AND Pin1ADVD AND Pin2RETD
							AND Pin3RETD AND Pin4ADVD AND Pin5RETD AND Pin6RETD AND Pin7RETD AND Pin8ADVD
							AND Slide1ADVD AND Slide2ADVD AND Slide3ADVD AND Slide4ADVD AND Slide5ADVD
							AND Slide6ADVD AND Slide7ADVD AND Slide8ADVD AND Slide9ADVD AND Slide10ADVD
							AND Slide11ADVD AND Slide12ADVD AND Slide13ADVD AND Slide14ADVD AND Slide15ADVD;
	END_IF
				
	Tool_At_Weld.1:= FALSE;
	Tool_At_Weld.2:= FALSE;
	Tool_At_Weld.3:= FALSE;
	Tool_At_Weld.4:= FALSE;


	IF ((Model_ID =1) OR (Model_ID=8) OR (Model_ID =2) OR (Model_ID=9)) THEN
		
				Tool_At_Unload.0:= Clamp1ADVD AND Clamp2ADVD AND Clamp3RETD AND Clamp4ADVD AND Clamp5RETD
							AND Clamp6RETD AND Clamp7ADVD AND Clamp8RETD AND Clamp9RETD AND Clamp10RETD
							AND Clamp11ADVD AND Clamp12RETD AND Clamp13ADVD AND Clamp14ADVD AND Clamp15ADVD
							AND Clamp16ADVD AND Clamp17ADVD AND Clamp18ADVD AND Clamp19ADVD AND Clamp20RETD
							AND Clamp21RETD AND Clamp22RETD AND Clamp23RETD AND Clamp24RETD AND Clamp25RETD
							AND Clamp26RETD AND Clamp27RETD AND Clamp28RETD AND Clamp29ADVD AND Clamp30RETD
							AND Clamp31RETD AND Clamp32ADVD AND Clamp33ADVD AND Clamp34RETD AND Clamp35ADVD
							AND Clamp36RETD AND Clamp37ADVD AND Clamp38RETD AND Pin1RETD AND Pin2RETD
							AND Pin3RETD AND Pin4RETD AND Pin5RETD AND Pin6RETD AND Pin7RETD AND Pin8RETD
							AND Slide1RETD AND Slide2RETD AND Slide3RETD AND Slide4ADVD AND Slide5RETD
							AND Slide6RETD AND Slide7ADVD AND Slide8ADVD AND Slide9RETD AND Slide10RETD
							AND Slide11ADVD AND Slide12RETD AND Slide13RETD AND Slide14RETD AND Slide15RETD;
							
		ELSIF ((Model_ID=3) OR (Model_ID=10)) THEN
			
				Tool_At_Unload.0:= Clamp1ADVD AND Clamp2ADVD AND Clamp3RETD AND Clamp4ADVD AND Clamp5RETD
							AND Clamp6RETD AND Clamp7RETD AND Clamp8ADVD AND Clamp9RETD AND Clamp10ADVD
							AND Clamp11ADVD AND Clamp12RETD AND Clamp13ADVD AND Clamp14ADVD AND Clamp15ADVD
							AND Clamp16ADVD AND Clamp17ADVD AND Clamp18ADVD AND Clamp19ADVD AND Clamp20RETD
							AND Clamp21RETD AND Clamp22RETD AND Clamp23RETD AND Clamp24ADVD AND Clamp25RETD
							AND Clamp26RETD AND Clamp27ADVD AND Clamp28RETD AND Clamp29ADVD AND Clamp30RETD
							AND Clamp31ADVD AND Clamp32ADVD AND Clamp33ADVD AND Clamp34RETD AND Clamp35RETD
							AND Clamp36RETD AND Clamp37ADVD AND Clamp38RETD AND Pin1RETD AND Pin2RETD
							AND Pin3RETD AND Pin4RETD AND Pin5RETD AND Pin6RETD AND Pin7RETD AND Pin8RETD
							AND Slide1RETD AND Slide2RETD AND Slide3RETD AND Slide4ADVD AND Slide5RETD
							AND Slide6RETD AND Slide7ADVD AND Slide8ADVD AND Slide9RETD AND Slide10RETD
							AND Slide11ADVD AND Slide12RETD AND Slide13RETD AND Slide14RETD AND Slide15RETD;
							
		ELSIF 			   (Model_ID=4) OR (Model_ID=5) OR (Model_ID=6) OR (Model_ID=7)
						OR (Model_ID=11) OR (Model_ID=12) OR (Model_ID=13) OR (Model_ID=14)
						OR (Model_ID=15) OR (Model_ID=16) OR (Model_ID=17) OR (Model_ID=18)
						OR (Model_ID=19) OR (Model_ID=20) OR (Model_ID=21) OR (Model_ID=22) THEN
			
				Tool_At_Unload.0:= Clamp1ADVD AND Clamp2ADVD AND Clamp3RETD AND Clamp4ADVD AND Clamp5RETD
							AND Clamp6RETD AND Clamp7ADVD AND Clamp8RETD AND Clamp9RETD AND Clamp10RETD
							AND Clamp11ADVD AND Clamp12RETD AND Clamp13ADVD AND Clamp14ADVD AND Clamp15ADVD
							AND Clamp16ADVD AND Clamp17ADVD AND Clamp18ADVD AND Clamp19ADVD AND Clamp20RETD
							AND Clamp21RETD AND Clamp22RETD AND Clamp23RETD AND Clamp24RETD AND Clamp25RETD
							AND Clamp26RETD AND Clamp27RETD AND Clamp28RETD AND Clamp29ADVD AND Clamp30RETD
							AND Clamp31RETD AND Clamp32ADVD AND Clamp33ADVD AND Clamp34RETD AND Clamp35ADVD
							AND Clamp36RETD AND Clamp37ADVD AND Clamp38RETD AND Pin1RETD AND Pin2RETD
							AND Pin3RETD AND Pin4RETD AND Pin5RETD AND Pin6RETD AND Pin7RETD AND Pin8RETD
							AND Slide1RETD AND Slide2RETD AND Slide3RETD AND Slide4ADVD AND Slide5RETD
							AND Slide6RETD AND Slide7ADVD AND Slide8ADVD AND Slide9RETD AND Slide10RETD
							AND Slide11ADVD AND Slide12RETD AND Slide13RETD AND Slide14RETD AND Slide15RETD;
	END_IF
	(*After Robot Repo 89*)			
	IF ((Model_ID =1) OR (Model_ID=8) OR (Model_ID =2) OR (Model_ID=9)) THEN
		
				Tool_At_Unload.1:= Clamp1ADVD AND Clamp2ADVD AND Clamp3RETD AND Clamp4RETD AND Clamp5RETD
							AND Clamp6RETD AND Clamp7RETD AND Clamp8RETD AND Clamp9RETD AND Clamp10RETD
							AND Clamp11RETD AND Clamp12RETD AND Clamp13ADVD AND Clamp14ADVD AND Clamp15ADVD
							AND Clamp16ADVD AND Clamp17ADVD AND Clamp18ADVD AND Clamp19ADVD AND Clamp20RETD
							AND Clamp21RETD AND Clamp22RETD AND Clamp23RETD AND Clamp24RETD AND Clamp25RETD
							AND Clamp26RETD AND Clamp27RETD AND Clamp28RETD AND Clamp29RETD AND Clamp30RETD
							AND Clamp31RETD AND Clamp32ADVD AND Clamp33RETD AND Clamp34RETD AND Clamp35RETD
							AND Clamp36RETD AND Clamp37ADVD AND Clamp38RETD AND Pin1RETD AND Pin2RETD
							AND Pin3RETD AND Pin4RETD AND Pin5RETD AND Pin6RETD AND Pin7RETD AND Pin8RETD
							AND Slide1RETD AND Slide2RETD AND Slide3RETD AND Slide4RETD AND Slide5RETD
							AND Slide6RETD AND Slide7ADVD AND Slide8RETD AND Slide9RETD AND Slide10RETD
							AND Slide11RETD AND Slide12RETD AND Slide13RETD AND Slide14RETD AND Slide15RETD;
							
		ELSIF ((Model_ID=3) OR (Model_ID=10)) THEN
			
				Tool_At_Unload.1:= Clamp1ADVD AND Clamp2ADVD AND Clamp3RETD AND Clamp4RETD AND Clamp5RETD
							AND Clamp6RETD AND Clamp7RETD AND Clamp8ADVD AND Clamp9RETD AND Clamp10ADVD
							AND Clamp11RETD AND Clamp12RETD AND Clamp13ADVD AND Clamp14ADVD AND Clamp15ADVD
							AND Clamp16ADVD AND Clamp17ADVD AND Clamp18ADVD AND Clamp19ADVD AND Clamp20RETD
							AND Clamp21RETD AND Clamp22RETD AND Clamp23RETD AND Clamp24ADVD AND Clamp25RETD
							AND Clamp26RETD AND Clamp27ADVD AND Clamp28RETD AND Clamp29RETD AND Clamp30RETD
							AND Clamp31ADVD AND Clamp32ADVD AND Clamp33RETD AND Clamp34RETD AND Clamp35RETD
							AND Clamp36RETD AND Clamp37ADVD AND Clamp38RETD AND Pin1RETD AND Pin2RETD
							AND Pin3RETD AND Pin4RETD AND Pin5RETD AND Pin6RETD AND Pin7RETD AND Pin8RETD
							AND Slide1RETD AND Slide2RETD AND Slide3RETD AND Slide4RETD AND Slide5RETD
							AND Slide6RETD AND Slide7ADVD AND Slide8RETD AND Slide9RETD AND Slide10RETD
							AND Slide11RETD AND Slide12RETD AND Slide13RETD AND Slide14RETD AND Slide15RETD;
							
		ELSIF 			   (Model_ID=4) OR (Model_ID=5) OR (Model_ID=6) OR (Model_ID=7)
						OR (Model_ID=11) OR (Model_ID=12) OR (Model_ID=13) OR (Model_ID=14)
						OR (Model_ID=15) OR (Model_ID=16) OR (Model_ID=17) OR (Model_ID=18)
						OR (Model_ID=19) OR (Model_ID=20) OR (Model_ID=21) OR (Model_ID=22) THEN
			
				Tool_At_Unload.1:= Clamp1ADVD AND Clamp2ADVD AND Clamp3RETD AND Clamp4RETD AND Clamp5RETD
							AND Clamp6RETD AND Clamp7RETD AND Clamp8RETD AND Clamp9RETD AND Clamp10RETD
							AND Clamp11RETD AND Clamp12RETD AND Clamp13ADVD AND Clamp14ADVD AND Clamp15ADVD
							AND Clamp16ADVD AND Clamp17ADVD AND Clamp18ADVD AND Clamp19ADVD AND Clamp20RETD
							AND Clamp21RETD AND Clamp22RETD AND Clamp23RETD AND Clamp24RETD AND Clamp25RETD
							AND Clamp26RETD AND Clamp27RETD AND Clamp28RETD AND Clamp29RETD AND Clamp30RETD
							AND Clamp31RETD AND Clamp32ADVD AND Clamp33RETD AND Clamp34RETD AND Clamp35RETD
							AND Clamp36RETD AND Clamp37ADVD AND Clamp38RETD AND Pin1RETD AND Pin2RETD
							AND Pin3RETD AND Pin4RETD AND Pin5RETD AND Pin6RETD AND Pin7RETD AND Pin8RETD
							AND Slide1RETD AND Slide2RETD AND Slide3RETD AND Slide4RETD AND Slide5RETD
							AND Slide6RETD AND Slide7ADVD AND Slide8RETD AND Slide9RETD AND Slide10RETD
							AND Slide11RETD AND Slide12RETD AND Slide13RETD AND Slide14RETD AND Slide15RETD;
	END_IF
	
	Tool_At_Unload.2:= FALSE;
	Tool_At_Unload.3:= FALSE;
	Tool_At_Unload.4:= FALSE;

(*end*)
END_ACTION

ACTION Tool_VBSeq_Repos:
(*+++++++++++THIS AREA IS CUSTOM PER INSTALLATION AND WILL HAVE TO BE MODIFIED PER +++++++++++++*)
(*+++++++++++THIS AREA IS CUSTOM PER INSTALLATION AND WILL HAVE TO BE MODIFIED PER +++++++++++++*)

(*!!!!!!!!!!!!!!!!!!!!!!!!!!!!!!!!!!!!!!!!!! Tool Motion Control !!!!!!!!!!!!!!!!!!!!!!!!!!!!!!!*)

(*----------------------------------------- Camp / Unclamp Steps -------------------------------*)

(*$$$$$$$$$$$$$$$$$$$$$$$$$$$$$$$$$$ Develop Clamp and Unclamp Interlocks $$$$$$$$$$$$$$$$$$$$$$*)
(* Note: This is one method to create valve bank commands for clamp and unclamp sequencing you are welcome to use the direct method as well*)

(*Start Clamp Sequence*)	
	
	(*First Stage Clamping*) (*V10, V11, V14, V15 ADV, IF Model 543, V19 ADV*)
		Clamp_Step.0:= Auto_Run AND (NOT Welding_Complete OR (Cycle_Complete AND NOT Tool_At_Home)) AND NOT All_Sensors_Off;

	(*Second Stage Clamping*)	(*V12, V13 ADV, IF Model 543, V20, V21 ADV*)
		(*504*)
			IF ((Model_ID=1) OR (Model_ID=8)) THEN
						Clamp_Step.1:=  Clamp_Step.0 AND 
										(*V10*)
										(Slide4ADVD AND Slide8ADVD AND Slide11ADVD)
										(*V11*)
										AND (Slide6ADVD)
										(*V14*)
										AND (Slide1ADVD AND Slide2ADVD AND Slide14ADVD AND Slide15ADVD)
										(*V15*)
										AND (Pin1ADVD AND Pin4ADVD AND Pin8ADVD);
		(*524*)						
				ELSIF ((Model_ID=2) OR (Model_ID=9)) THEN
						Clamp_Step.1:=  Clamp_Step.0 AND 
										(*V10*)
										(Slide4ADVD AND Slide8ADVD AND Slide11ADVD)
										(*V11*)
										AND (Slide6ADVD)
										(*V14*)
										AND (Slide1ADVD AND Slide2ADVD AND Slide14ADVD AND Slide15ADVD)
										(*V15*)
										AND (Pin1ADVD AND Pin4ADVD AND Pin8ADVD);
		(*543*)						
				ELSIF ((Model_ID=3) OR (Model_ID=10)) THEN
						Clamp_Step.1:=  Clamp_Step.0 AND 
										(*V10*)
										(Slide4ADVD AND Slide8ADVD AND Slide11ADVD)
										(*V11*)
										AND (Slide6ADVD)
										(*V14*)
										AND (Slide1ADVD AND Slide2ADVD AND Slide14ADVD AND Slide15ADVD)
										(*V15*)
										AND (Pin1ADVD AND Pin4ADVD AND Pin8ADVD)
										(*V19*)
										AND (Pin2ADVD AND Pin5ADVD AND Pin7ADVD);
		(*526*)						
				ELSIF ((Model_ID=4) OR (Model_ID=11) OR (Model_ID=15) OR (Model_ID=19)) THEN
						Clamp_Step.1:=  Clamp_Step.0 AND 
										(*V10*)
										(Slide4ADVD AND Slide8ADVD AND Slide11ADVD)
										(*V11*)
										AND (Slide6ADVD)
										(*V14*)
										AND (Slide1ADVD AND Slide2ADVD AND Slide14ADVD AND Slide15ADVD)
										(*V15*)
										AND (Pin1ADVD AND Pin4ADVD AND Pin8ADVD);
		(*536*)						
				ELSIF ((Model_ID=5) OR (Model_ID=12) OR (Model_ID=16) OR (Model_ID=20)) THEN
						Clamp_Step.1:=  Clamp_Step.0 AND 
										(*V10*)
										(Slide4ADVD AND Slide8ADVD AND Slide11ADVD)
										(*V11*)
										AND (Slide6ADVD)
										(*V14*)
										AND (Slide1ADVD AND Slide2ADVD AND Slide14ADVD AND Slide15ADVD)
										(*V15*)
										AND (Pin1ADVD AND Pin4ADVD AND Pin8ADVD);
		(*550*)						
				ELSIF ((Model_ID=6) OR (Model_ID=13) OR (Model_ID=17) OR (Model_ID=21)) THEN
						Clamp_Step.1:=  Clamp_Step.0 AND 
										(*V10*)
										(Slide4ADVD AND Slide8ADVD AND Slide11ADVD)
										(*V11*)
										AND (Slide6ADVD)
										(*V14*)
										AND (Slide1ADVD AND Slide2ADVD AND Slide14ADVD AND Slide15ADVD)
										(*V15*)
										AND (Pin1ADVD AND Pin4ADVD AND Pin8ADVD);
		(*571*)						
				ELSIF ((Model_ID=7) OR (Model_ID=14) OR (Model_ID=18) OR (Model_ID=22)) THEN
						Clamp_Step.1:=  Clamp_Step.0 AND 
										(*V10*)
										(Slide4ADVD AND Slide8ADVD AND Slide11ADVD)
										(*V11*)
										AND (Slide6ADVD)
										(*V14*)
										AND (Slide1ADVD AND Slide2ADVD AND Slide14ADVD AND Slide15ADVD)
										(*V15*)
										AND (Pin1ADVD AND Pin4ADVD AND Pin8ADVD);
			END_IF

	(*Third Stage Clamping*)	(*V1-V7 ADV, IF Model 504, 524, V8 ADV, IF Model 526, 536, 550, 571, V9 ADV, IF Model 543, V18 ADV*)
		(*504*)
			IF ((Model_ID=1) OR (Model_ID=8)) THEN
						Clamp_Step.2:= Clamp_Step.1 AND 
										(*V12*)
										(Slide7ADVD)
										(*V13*)
										AND (Slide10ADVD);
		(*524*)						
				ELSIF ((Model_ID=2) OR (Model_ID=9)) THEN
						Clamp_Step.2:= Clamp_Step.1 AND 
										(*V12*)
										(Slide7RETD)
										(*V13*)
										AND (Slide10ADVD);
		(*543*)				
				ELSIF ((Model_ID=3) OR (Model_ID=10)) THEN
						Clamp_Step.2:= Clamp_Step.1 AND 
										(*V12*)
										(Slide7ADVD)
										(*V13*)
										AND (Slide10ADVD)
										(*V20*)
										AND (Clamp8ADVD AND Clamp24ADVD AND Clamp31ADVD)
										(*V21*)
										AND (Clamp10ADVD AND Clamp27ADVD);
		(*526*)
				ELSIF ((Model_ID=4) OR (Model_ID=11) OR (Model_ID=15) OR (Model_ID=19)) THEN
						Clamp_Step.2:= Clamp_Step.1 AND 
										(*V12*)
										(Slide7RETD)
										(*V13*)
										AND (Slide10ADVD);
		(*536*)						
				ELSIF ((Model_ID=5) OR (Model_ID=12) OR (Model_ID=16) OR (Model_ID=20)) THEN
						Clamp_Step.2:= Clamp_Step.1 AND 
										(*V12*)
										(Slide7RETD)
										(*V13*)
										AND (Slide10ADVD);
		(*550*)						
				ELSIF ((Model_ID=6) OR (Model_ID=13) OR (Model_ID=17) OR (Model_ID=21)) THEN
						Clamp_Step.2:= Clamp_Step.1 AND 
										(*V12*)
										(Slide7RETD)
										(*V13*)
										AND (Slide10ADVD);
		(*571*)						
				ELSIF ((Model_ID=7) OR (Model_ID=14) OR (Model_ID=18) OR (Model_ID=22)) THEN
						Clamp_Step.2:= Clamp_Step.1 AND 
										(*V12*)
										(Slide7RETD)
										(*V13*)
										AND (Slide10ADVD);
			END_IF
														
	(*Forth Stage Clamping*)	(*Fire QAs - V17*)
		(*504*)	
			IF ((Model_ID=1) OR (Model_ID=8)) THEN
						Clamp_Step.3:= Clamp_Step.2 AND 
										(*V1*)
										(Clamp1ADVD AND Clamp2ADVD AND Clamp32ADVD AND Clamp37ADVD)
										(*V2*)
										AND (Clamp13ADVD AND Clamp14ADVD AND Clamp15ADVD)
										(*V3*)
										AND (Clamp16ADVD AND Clamp17ADVD AND Clamp18ADVD AND Clamp19ADVD)
										(*V4*)
										AND (Clamp3ADVD AND Clamp12ADVD AND Clamp20ADVD AND Clamp28ADVD AND Clamp34ADVD)
										(*V5*)
										AND (Clamp4ADVD AND Clamp11ADVD AND Clamp21ADVD AND Clamp29ADVD AND Clamp33ADVD)
										(*V6*)
										AND (Clamp6ADVD AND Clamp9ADVD AND Clamp30ADVD AND Clamp36ADVD)
										(*V7*)
										AND (Clamp7ADVD AND Clamp35ADVD)
										(*V8*)
										AND (Clamp22ADVD AND Clamp26ADVD);
		(*524*)						
				ELSIF ((Model_ID=2) OR (Model_ID=9)) THEN
						Clamp_Step.3:= Clamp_Step.2 AND 
										(*V1*)
										(Clamp1ADVD AND Clamp2ADVD AND Clamp32ADVD AND Clamp37ADVD)
										(*V2*)
										AND (Clamp13ADVD AND Clamp14ADVD AND Clamp15ADVD)
										(*V3*)
										AND (Clamp16ADVD AND Clamp17ADVD AND Clamp18ADVD AND Clamp19ADVD)
										(*V4*)
										AND (Clamp3ADVD AND Clamp12ADVD AND Clamp20ADVD AND Clamp28ADVD AND Clamp34ADVD)
										(*V5*)
										AND (Clamp4ADVD AND Clamp11ADVD AND Clamp21ADVD AND Clamp29ADVD AND Clamp33ADVD)
										(*V6*)
										AND (Clamp6ADVD AND Clamp9ADVD AND Clamp30ADVD AND Clamp36ADVD)
										(*V7*)
										AND (Clamp7ADVD AND Clamp35ADVD)
										(*V8*)
										AND (Clamp22ADVD AND Clamp26ADVD);								
		(*543*)						
				ELSIF ((Model_ID=3) OR (Model_ID=10)) THEN
						Clamp_Step.3:= Clamp_Step.2 AND 
										(*V1*)
										(Clamp1ADVD AND Clamp2ADVD AND Clamp32ADVD AND Clamp37ADVD)
										(*V2*)
										AND (Clamp13ADVD AND Clamp14ADVD AND Clamp15ADVD)
										(*V3*)
										AND (Clamp16ADVD AND Clamp17ADVD AND Clamp18ADVD AND Clamp19ADVD)
										(*V4*)
										AND (Clamp3ADVD AND Clamp12ADVD AND Clamp20ADVD AND Clamp28ADVD AND Clamp34ADVD)
										(*V5*)
										AND (Clamp4ADVD AND Clamp11ADVD AND Clamp21ADVD AND Clamp29ADVD AND Clamp33ADVD)
										(*V6*)
										AND (Clamp6ADVD AND Clamp9ADVD AND Clamp30ADVD AND Clamp36ADVD)
										(*V7*)
										AND (Clamp7ADVD AND Clamp35ADVD)
										(*V18*)
										AND (Pin3ADVD AND Pin6ADVD);
		(*526*)						
				ELSIF ((Model_ID=4) OR (Model_ID=11) OR (Model_ID=15) OR (Model_ID=19)) THEN
						Clamp_Step.3:= Clamp_Step.2 AND 
										(*V1*)
										(Clamp1ADVD AND Clamp2ADVD AND Clamp32ADVD AND Clamp37ADVD)
										(*V2*)
										AND (Clamp13ADVD AND Clamp14ADVD AND Clamp15ADVD)
										(*V3*)
										AND (Clamp16ADVD AND Clamp17ADVD AND Clamp18ADVD AND Clamp19ADVD)
										(*V4*)
										AND (Clamp3ADVD AND Clamp12ADVD AND Clamp20ADVD AND Clamp28ADVD AND Clamp34ADVD)
										(*V5*)
										AND (Clamp4ADVD AND Clamp11ADVD AND Clamp21ADVD AND Clamp29ADVD AND Clamp33ADVD)
										(*V6*)
										AND (Clamp6ADVD AND Clamp9ADVD AND Clamp30ADVD AND Clamp36ADVD)
										(*V7*)
										AND (Clamp7ADVD AND Clamp35ADVD)
										(*V9*)
										AND (Clamp23ADVD AND Clamp25ADVD);
		(*536*)						
				ELSIF ((Model_ID=5) OR (Model_ID=12) OR (Model_ID=16) OR (Model_ID=20)) THEN
						Clamp_Step.3:= Clamp_Step.2 AND 
										(*V1*)
										(Clamp1ADVD AND Clamp2ADVD AND Clamp32ADVD AND Clamp37ADVD)
										(*V2*)
										AND (Clamp13ADVD AND Clamp14ADVD AND Clamp15ADVD)
										(*V3*)
										AND (Clamp16ADVD AND Clamp17ADVD AND Clamp18ADVD AND Clamp19ADVD)
										(*V4*)
										AND (Clamp3ADVD AND Clamp12ADVD AND Clamp20ADVD AND Clamp28ADVD AND Clamp34ADVD)
										(*V5*)
										AND (Clamp4ADVD AND Clamp11ADVD AND Clamp21ADVD AND Clamp29ADVD AND Clamp33ADVD)
										(*V6*)
										AND (Clamp6ADVD AND Clamp9ADVD AND Clamp30ADVD AND Clamp36ADVD)
										(*V7*)
										AND (Clamp7ADVD AND Clamp35ADVD)
										(*V9*)
										AND (Clamp23ADVD AND Clamp25ADVD);
		(*550*)
				ELSIF ((Model_ID=6) OR (Model_ID=13) OR (Model_ID=17) OR (Model_ID=21)) THEN
						Clamp_Step.3:= Clamp_Step.2 AND 
										(*V1*)
										(Clamp1ADVD AND Clamp2ADVD AND Clamp32ADVD AND Clamp37ADVD)
										(*V2*)
										AND (Clamp13ADVD AND Clamp14ADVD AND Clamp15ADVD)
										(*V3*)
										AND (Clamp16ADVD AND Clamp17ADVD AND Clamp18ADVD AND Clamp19ADVD)
										(*V4*)
										AND (Clamp3ADVD AND Clamp12ADVD AND Clamp20ADVD AND Clamp28ADVD AND Clamp34ADVD)
										(*V5*)
										AND (Clamp4ADVD AND Clamp11ADVD AND Clamp21ADVD AND Clamp29ADVD AND Clamp33ADVD)
										(*V6*)
										AND (Clamp6ADVD AND Clamp9ADVD AND Clamp30ADVD AND Clamp36ADVD)
										(*V7*)
										AND (Clamp7ADVD AND Clamp35ADVD)
										(*V9*)
										AND (Clamp23ADVD AND Clamp25ADVD);
		(*571*)
				ELSIF ((Model_ID=7) OR (Model_ID=14) OR (Model_ID=18) OR (Model_ID=22)) THEN
						Clamp_Step.3:= Clamp_Step.2 AND 
										(*V1*)
										(Clamp1ADVD AND Clamp2ADVD AND Clamp32ADVD AND Clamp37ADVD)
										(*V2*)
										AND (Clamp13ADVD AND Clamp14ADVD AND Clamp15ADVD)
										(*V3*)
										AND (Clamp16ADVD AND Clamp17ADVD AND Clamp18ADVD AND Clamp19ADVD)
										(*V4*)
										AND (Clamp3ADVD AND Clamp12ADVD AND Clamp20ADVD AND Clamp28ADVD AND Clamp34ADVD)
										(*V5*)
										AND (Clamp4ADVD AND Clamp11ADVD AND Clamp21ADVD AND Clamp29ADVD AND Clamp33ADVD)
										(*V6*)
										AND (Clamp6ADVD AND Clamp9ADVD AND Clamp30ADVD AND Clamp36ADVD)
										(*V7*)
										AND (Clamp7ADVD AND Clamp35ADVD)
										(*V9*)
										AND (Clamp23ADVD AND Clamp25ADVD);								
			END_IF
	
	
	(*Fifth Stage Clamping*)	(*V16 ADV*)
			(*QA Check All Models*)
				Clamp_Step.4:= Clamp_Step.3 (*AND
					CheckQA1FB.QAcheck_OK*); (*Positions are off currently - AB*)
	
	
(*Start Unclamp Sequence*)
	(*First Stage Unclamping*)	(*V11, V13, V15, V16 RET, IF Model 543, V18, V19 RET*)
		Unclamp_Step.0:= (Welding_Complete AND TurnTableB_At_Robot AND NOT (MAIN.R1.Task_ID_Ack=Sweep_Fix01) AND NOT (MAIN.R1.Task_ID_Ack=Sweep_Fix03) AND NOT Cycle_Complete);
	
	(*Second Stage Unclamping*)	(*V4, V6, V14 RET, IF Model 504, 524, V8 RET, IF Model 526, 536, 550, 571, V9 RET*)
		(*504*)
			IF ((Model_ID=1) OR (Model_ID=8)) THEN
							Unclamp_Step.1:= Unclamp_Step.0 AND 
											(*V11*)
											(Slide6RETD)
											(*V13*)
											AND (Slide10RETD)
											(*V15*)
											AND (Pin1RETD AND Pin4RETD AND Pin8RETD)
											(*V16*)
											AND (Clamp5RETD AND Clamp38RETD AND Slide3RETD AND Slide5RETD AND Slide9RETD AND Slide12RETD AND Slide13RETD);
		(*524*)								
				ELSIF ((Model_ID=2) OR (Model_ID=9)) THEN
							Unclamp_Step.1:= Unclamp_Step.0 AND 
											(*V11*)
											(Slide6RETD)
											(*V13*)
											AND (Slide10RETD)
											(*V15*)
											AND (Pin1RETD AND Pin4RETD AND Pin8RETD)
											(*V16*)
											AND (Clamp5RETD AND Clamp38RETD AND Slide3RETD AND Slide5RETD AND Slide9RETD AND Slide12RETD AND Slide13RETD);

		(*543*)									
				ELSIF ((Model_ID=3) OR (Model_ID=10)) THEN
							Unclamp_Step.1:= Unclamp_Step.0 AND 
											(*V11*)
											(Slide6RETD)
											(*V13*)
											AND (Slide10RETD)
											(*V15*)
											AND (Pin1RETD AND Pin4RETD AND Pin8RETD)
											(*V16*)
											AND (Clamp5RETD AND Clamp38RETD AND Slide3RETD AND Slide5RETD AND Slide9RETD AND Slide12RETD AND Slide13RETD)
											(*V18*)
											AND (Pin3RETD AND Pin6RETD)
											(*V19*)
											AND (Pin2RETD AND Pin5RETD AND Pin7RETD);
		(*526*)									
				ELSIF ((Model_ID=4) OR (Model_ID=11) OR (Model_ID=15) OR (Model_ID=19)) THEN
							Unclamp_Step.1:= Unclamp_Step.0 AND 
											(*V11*)
											(Slide6RETD)
											(*V13*)
											AND (Slide10RETD)
											(*V15*)
											AND (Pin1RETD AND Pin4RETD AND Pin8RETD)
											(*V16*)
											AND (Clamp5RETD AND Clamp38RETD AND Slide3RETD AND Slide5RETD AND Slide9RETD AND Slide12RETD AND Slide13RETD);
		(*536*)
				ELSIF ((Model_ID=5) OR (Model_ID=12) OR (Model_ID=16) OR (Model_ID=20)) THEN
							Unclamp_Step.1:= Unclamp_Step.0 AND 
											(*V11*)
											(Slide6RETD)
											(*V13*)
											AND (Slide10RETD)
											(*V15*)
											AND (Pin1RETD AND Pin4RETD AND Pin8RETD)
											(*V16*)
											AND (Clamp5RETD AND Clamp38RETD AND Slide3RETD AND Slide5RETD AND Slide9RETD AND Slide12RETD AND Slide13RETD);
		(*550*)
				ELSIF ((Model_ID=6) OR (Model_ID=13) OR (Model_ID=17) OR (Model_ID=21)) THEN
							Unclamp_Step.1:= Unclamp_Step.0 AND 
											(*V11*)
											(Slide6RETD)
											(*V13*)
											AND (Slide10RETD)
											(*V15*)
											AND (Pin1RETD AND Pin4RETD AND Pin8RETD)
											(*V16*)
											AND (Clamp5RETD AND Clamp38RETD AND Slide3RETD AND Slide5RETD AND Slide9RETD AND Slide12RETD AND Slide13RETD);
		(*571*)
				ELSIF ((Model_ID=7) OR (Model_ID=14) OR (Model_ID=18) OR (Model_ID=22)) THEN
							Unclamp_Step.1:= Unclamp_Step.0 AND 
											(*V11*)
											(Slide6RETD)
											(*V13*)
											AND (Slide10RETD)
											(*V15*)
											AND (Pin1RETD AND Pin4RETD AND Pin8RETD)
											(*V16*)
											AND (Clamp5RETD AND Clamp38RETD AND Slide3RETD AND Slide5RETD AND Slide9RETD AND Slide12RETD AND Slide13RETD);											
			END_IF									

									
	(*Third Stage Unclamping*)	(*V5, V10 RET, IF NOT Model 543, V7 RET*)
		(*504*)
			IF ((Model_ID=1) OR (Model_ID=8)) THEN
							Unclamp_Step.2:= Unclamp_Step.1 AND 
											(*V4*)
											(Clamp3RETD AND Clamp12RETD AND Clamp20RETD AND Clamp28RETD AND Clamp34RETD)
											(*V6*)
											AND (Clamp6RETD AND Clamp9RETD AND Clamp30RETD AND Clamp36RETD)
											(*V14*)
											AND (Slide1RETD AND Slide2RETD AND Slide14RETD AND Slide15RETD)
											(*V8*)
											AND (Clamp22RETD AND Clamp26RETD);
		(*524*)											
				ELSIF ((Model_ID=2) OR (Model_ID=9)) THEN
							Unclamp_Step.2:= Unclamp_Step.1 AND 
											(*V4*)
											(Clamp3RETD AND Clamp12RETD AND Clamp20RETD AND Clamp28RETD AND Clamp34RETD)
											(*V6*)
											AND (Clamp6RETD AND Clamp9RETD AND Clamp30RETD AND Clamp36RETD)
											(*V14*)
											AND (Slide1RETD AND Slide2RETD AND Slide14RETD AND Slide15RETD)
											(*V8*)
											AND (Clamp22RETD AND Clamp26RETD);
		(*543*)									
				ELSIF ((Model_ID=3) OR (Model_ID=10)) THEN
							Unclamp_Step.2:= Unclamp_Step.1 AND 
											(*V4*)
											(Clamp3RETD AND Clamp12RETD AND Clamp20RETD AND Clamp28RETD AND Clamp34RETD)
											(*V6*)
											AND (Clamp6RETD AND Clamp9RETD AND Clamp30RETD AND Clamp36RETD)
											(*V14*)
											AND (Slide1RETD AND Slide2RETD AND Slide14RETD AND Slide15RETD);
		(*526*)									
				ELSIF ((Model_ID=4) OR (Model_ID=11) OR (Model_ID=15) OR (Model_ID=19)) THEN
							Unclamp_Step.2:= Unclamp_Step.1 AND 
											(*V4*)
											(Clamp3RETD AND Clamp12RETD AND Clamp20RETD AND Clamp28RETD AND Clamp34RETD)
											(*V6*)
											AND (Clamp6RETD AND Clamp9RETD AND Clamp30RETD AND Clamp36RETD)
											(*V14*)
											AND (Slide1RETD AND Slide2RETD AND Slide14RETD AND Slide15RETD)
											(*V9*)
											AND (Clamp23RETD AND Clamp25RETD);
		(*536*)									
				ELSIF ((Model_ID=5) OR (Model_ID=12) OR (Model_ID=16) OR (Model_ID=20)) THEN
							Unclamp_Step.2:= Unclamp_Step.1 AND 
											(*V4*)
											(Clamp3RETD AND Clamp12RETD AND Clamp20RETD AND Clamp28RETD AND Clamp34RETD)
											(*V6*)
											AND (Clamp6RETD AND Clamp9RETD AND Clamp30RETD AND Clamp36RETD)
											(*V14*)
											AND (Slide1RETD AND Slide2RETD AND Slide14RETD AND Slide15RETD)
											(*V9*)
											AND (Clamp23RETD AND Clamp25RETD);
		(*550*)
				ELSIF  ((Model_ID=6) OR (Model_ID=13) OR (Model_ID=17) OR (Model_ID=21)) THEN
							Unclamp_Step.2:= Unclamp_Step.1 AND 
											(*V4*)
											(Clamp3RETD AND Clamp12RETD AND Clamp20RETD AND Clamp28RETD AND Clamp34RETD)
											(*V6*)
											AND (Clamp6RETD AND Clamp9RETD AND Clamp30RETD AND Clamp36RETD)
											(*V14*)
											AND (Slide1RETD AND Slide2RETD AND Slide14RETD AND Slide15RETD)
											(*V9*)
											AND (Clamp23RETD AND Clamp25RETD);
		(*571*)
				ELSIF ((Model_ID=7) OR (Model_ID=14) OR (Model_ID=18) OR (Model_ID=22)) THEN
							Unclamp_Step.2:= Unclamp_Step.1 AND 
											(*V4*)
											(Clamp3RETD AND Clamp12RETD AND Clamp20RETD AND Clamp28RETD AND Clamp34RETD)
											(*V6*)
											AND (Clamp6RETD AND Clamp9RETD AND Clamp30RETD AND Clamp36RETD)
											(*V14*)
											AND (Slide1RETD AND Slide2RETD AND Slide14RETD AND Slide15RETD)
											(*V9*)
											AND (Clamp23RETD AND Clamp25RETD);										
			END_IF				
					
	(*Fourth Stage Unclamping*)	(*V1-V3, V12 RET, IF Model 543, V20, V21 RET*)
		(*504*)
			IF NOT ((Model_ID=1) OR (Model_ID=8)) THEN
							Unclamp_Step.3:= Unclamp_Step.2 AND 
											(*V5*)
											(Clamp4RETD AND Clamp11RETD AND Clamp21RETD AND Clamp29RETD AND Clamp33RETD)
											(*V10*)
											AND (Slide4RETD AND Slide8RETD AND Slide11RETD)
											(*V7*)
											AND (Clamp7RETD AND Clamp35RETD);
		(*524*)								
				ELSIF ((Model_ID=2) OR (Model_ID=9)) THEN
							Unclamp_Step.3:= Unclamp_Step.2 AND 
											(*V5*)
											(Clamp4RETD AND Clamp11RETD AND Clamp21RETD AND Clamp29RETD AND Clamp33RETD)
											(*V10*)
											AND (Slide4RETD AND Slide8RETD AND Slide11RETD)
											(*V7*)
											AND (Clamp7RETD AND Clamp35RETD);											
		(*543*)									
				ELSIF ((Model_ID=3) OR (Model_ID=10)) THEN
							Unclamp_Step.3:= Unclamp_Step.2 AND 
											(*V5*)
											(Clamp4RETD AND Clamp11RETD AND Clamp21RETD AND Clamp29RETD AND Clamp33RETD)
											(*V10*)
											AND (Slide4RETD AND Slide8RETD AND Slide11RETD);
		(*526*)
				ELSIF ((Model_ID=4) OR (Model_ID=11) OR (Model_ID=15) OR (Model_ID=19)) THEN
							Unclamp_Step.3:= Unclamp_Step.2 AND 
											(*V5*)
											(Clamp4RETD AND Clamp11RETD AND Clamp21RETD AND Clamp29RETD AND Clamp33RETD)
											(*V10*)
											AND (Slide4RETD AND Slide8RETD AND Slide11RETD)
											(*V7*)
											AND (Clamp7RETD AND Clamp35RETD);
		(*536*)
				ELSIF ((Model_ID=5) OR (Model_ID=12) OR (Model_ID=16) OR (Model_ID=20)) THEN
							Unclamp_Step.3:= Unclamp_Step.2 AND 
											(*V5*)
											(Clamp4RETD AND Clamp11RETD AND Clamp21RETD AND Clamp29RETD AND Clamp33RETD)
											(*V10*)
											AND (Slide4RETD AND Slide8RETD AND Slide11RETD)
											(*V7*)
											AND (Clamp7RETD AND Clamp35RETD);
		(*550*)
				ELSIF ((Model_ID=6) OR (Model_ID=13) OR (Model_ID=17) OR (Model_ID=21)) THEN
							Unclamp_Step.3:= Unclamp_Step.2 AND 
											(*V5*)
											(Clamp4RETD AND Clamp11RETD AND Clamp21RETD AND Clamp29RETD AND Clamp33RETD)
											(*V10*)
											AND (Slide4RETD AND Slide8RETD AND Slide11RETD)
											(*V7*)
											AND (Clamp7RETD AND Clamp35RETD);
		(*571*)
				ELSIF ((Model_ID=7) OR (Model_ID=14) OR (Model_ID=18) OR (Model_ID=22)) THEN
							Unclamp_Step.3:= Unclamp_Step.2 AND 
											(*V5*)
											(Clamp4RETD AND Clamp11RETD AND Clamp21RETD AND Clamp29RETD AND Clamp33RETD)
											(*V10*)
											AND (Slide4RETD AND Slide8RETD AND Slide11RETD)
											(*V7*)
											AND (Clamp7RETD AND Clamp35RETD);					
			END_IF	

(*(*+++++++++++THIS AREA IS CUSTOM PER INSTALLATION AND WILL HAVE TO BE MODIFIED PER +++++++++++++*)
(*+++++++++++THIS AREA IS CUSTOM PER INSTALLATION AND WILL HAVE TO BE MODIFIED PER +++++++++++++*)


(*!!!!!!!!!!!!!!!!!!!!!!!!!!!!!!!!!!!!!!!!!! Tool Motion Control !!!!!!!!!!!!!!!!!!!!!!!!!!!!!!!*)

(*----------------------------------------- Clamp / Unclamp Steps -------------------------------*)

(*$$$$$$$$$$$$$$$$$$$$$$$$$$$$$$$$$$ Develop Clamp and Unclamp Interlocks $$$$$$$$$$$$$$$$$$$$$$*)
(* Note: This is one method to create valve bank commands for clamp and unclamp sequencing
you are welcome to use the direct method as well*)

	(*Start Clamp Sequence*)
	
	
	(*First Stage Clamping*) (*V10, V11, V14, V15 ADV, IF Model 543, V19 ADV*)
	Clamp_Step.0:= (Auto_Run AND NOT Welding_Complete AND TurntableB_At_Robot AND Load_Complete1) 
				OR
					(Valve1FB.SideB_Indicator AND Valve2FB.SideB_Indicator AND Valve3FB.SideB_Indicator 
					AND Valve12FB.SideB_Indicator (*AND All_Subs_Complete*) AND TurntableB_At_Robot);

	(*Second Stage Clamping*)	(*V6, V12, V13, V23 ADV, IF Model 543, V20, V21 ADV*)
	IF NOT (Model_ID=3) AND Load_Complete1 THEN
				Clamp_Step.1:=  Clamp_Step.0 AND 
								(*V10*)
								(Slide4ADVD AND Slide8ADVD AND Slide11ADVD)
								(*V11*)
								AND (Slide6ADVD)
								(*V14*)
								AND (Slide1ADVD AND Slide2ADVD AND Slide14ADVD AND Slide15ADVD)
								(*V15*)
								AND (Pin1ADVD AND Pin4ADVD AND Pin8ADVD);
		ELSIF (Model_ID=3) AND Load_Complete1 THEN
				Clamp_Step.1:=  Clamp_Step.0 AND 
								(*V10*)
								(Slide4ADVD AND Slide8ADVD AND Slide11ADVD)
								(*V11*)
								AND (Slide6ADVD)
								(*V14*)
								AND (Slide1ADVD AND Slide2ADVD AND Slide14ADVD AND Slide15ADVD)
								(*V15*)
								AND (Pin1ADVD AND Pin4ADVD AND Pin8ADVD)
								(*V19*)
								AND (Pin2ADVD AND Pin5ADVD AND Pin7ADVD);
		ELSE
			Clamp_Step.1:= FALSE;
	END_IF

	(*Third Stage Clamping*)	(*V1-V7 ADV, IF Model 504, 524, V8 ADV, IF Model 526, 536, 550, 571, V9 ADV, IF Model 543, V18 ADV*)
	IF (Model_ID<3) THEN
				Clamp_Step.2:= Clamp_Step.1 AND 
								(*V12*)
								(Slide7ADVD);
		ELSIF (Model_ID=3) THEN
				Clamp_Step.2:= Clamp_Step.1 AND 
								(*V12*)
								(Slide7ADVD)
								(*V13*)
								AND (Slide10RETD)
								(*V20*)
								AND (Clamp8ADVD AND Clamp24ADVD AND Clamp31ADVD)
								(*V21*)
								AND (Clamp10ADVD AND Clamp27ADVD);
		ELSIF (Model_ID>3) THEN
				Clamp_Step.2:= Clamp_Step.1 AND 
								(*V12*)
								(Slide7ADVD)
								(*V13*)
								AND (Slide10ADVD);
		ELSE
			Clamp_Step.2:= FALSE;
	END_IF
														
	(*Forth Stage Clamping*)	(*Fire QAs - V17*)
	IF (Model_ID<3) THEN
				Clamp_Step.3:= Clamp_Step.2 AND 
								(*V1*)
								(Clamp1ADVD AND Clamp2ADVD AND Clamp32ADVD AND Clamp37ADVD)
								(*V2*)
								AND (Clamp13ADVD AND Clamp14ADVD AND Clamp15ADVD)
								(*V3*)
								AND (Clamp16ADVD AND Clamp17ADVD AND Clamp18ADVD AND Clamp19ADVD)
								(*V4*)
								AND (Clamp3ADVD AND Clamp12ADVD AND Clamp20ADVD AND Clamp28ADVD AND Clamp34ADVD)
								(*V5*)
								AND (Clamp4ADVD AND Clamp11ADVD AND Clamp21ADVD AND Clamp29ADVD AND Clamp33ADVD)
								(*V6*)
								AND (Clamp6ADVD AND Clamp9ADVD AND Clamp30ADVD AND Clamp36ADVD)
								(*V7*)
								AND (Clamp7ADVD AND Clamp35ADVD)
								(*V8*)
								AND (Clamp22ADVD AND Clamp26ADVD);
		ELSIF (Model_ID=3) THEN
				Clamp_Step.3:= Clamp_Step.2 AND 
								(*V1*)
								(Clamp1ADVD AND Clamp2ADVD AND Clamp32ADVD AND Clamp37ADVD)
								(*V2*)
								AND (Clamp13ADVD AND Clamp14ADVD AND Clamp15ADVD)
								(*V3*)
								AND (Clamp16ADVD AND Clamp17ADVD AND Clamp18ADVD AND Clamp19ADVD)
								(*V4*)
								AND (Clamp3ADVD AND Clamp12ADVD AND Clamp20ADVD AND Clamp28ADVD AND Clamp34ADVD)
								(*V5*)
								AND (Clamp4ADVD AND Clamp11ADVD AND Clamp21ADVD AND Clamp29ADVD AND Clamp33ADVD)
								(*V6*)
								AND (Clamp6ADVD AND Clamp9ADVD AND Clamp30ADVD AND Clamp36ADVD)
								(*V18*)
								AND (Pin3ADVD AND Pin6ADVD);
		ELSIF (Model_ID>3) THEN
				Clamp_Step.3:= Clamp_Step.2 AND 
								(*V1*)
								(Clamp1ADVD AND Clamp2ADVD AND Clamp32ADVD AND Clamp37ADVD)
								(*V2*)
								AND (Clamp13ADVD AND Clamp14ADVD AND Clamp15ADVD)
								(*V3*)
								AND (Clamp16ADVD AND Clamp17ADVD AND Clamp18ADVD AND Clamp19ADVD)
								(*V4*)
								AND (Clamp3ADVD AND Clamp12ADVD AND Clamp20ADVD AND Clamp28ADVD AND Clamp34ADVD)
								(*V5*)
								AND (Clamp4ADVD AND Clamp11ADVD AND Clamp21ADVD AND Clamp29ADVD AND Clamp33ADVD)
								(*V6*)
								AND (Clamp6ADVD AND Clamp9ADVD AND Clamp30ADVD AND Clamp36ADVD)
								(*V7*)
								AND (Clamp7ADVD AND Clamp35ADVD)
								(*V9*)
								AND (Clamp23ADVD AND Clamp25ADVD);
		ELSE
			Clamp_Step.3:= FALSE;

	END_IF
	
	
	(*Fifth Stage Clamping*)	(*V16 ADV*)
	Clamp_Step.4:= Clamp_Step.3 AND
					CheckQA1FB.QAcheck_OK;
	
	
	
	
	(*Start Unclamp Sequence*)
	(*First Stage Unclamping*)	(*V11, V13, V15, V16 RET, IF Model 543, V18, V19 RET*)
	Unclamp_Step.0:= Welding_Complete AND TurntableA_At_Robot;
	
	(*Second Stage Unclamping*)	(*V4, V6, V14 RET, IF Model 504, 524, V8 RET, IF Model 526, 536, 550, 571, V9 RET*)
	IF NOT (Model_ID=3) THEN
					Unclamp_Step.1:= Unclamp_Step.0 AND 
									(*V11*)
									(Slide6RETD)
									(*V13*)
									AND (Slide10RETD)
									(*V15*)
									AND (Pin1RETD AND Pin4RETD AND Pin8RETD)
									(*V16*)
									AND (Clamp5RETD AND Clamp38RETD AND Slide3RETD AND Slide5RETD AND Slide9RETD AND Slide12RETD AND Slide13RETD);
									
		ELSIF (Model_ID=3) THEN
					Unclamp_Step.1:= Unclamp_Step.0 AND 
									(*V11*)
									(Slide6RETD)
									(*V13*)
									AND (Slide10RETD)
									(*V15*)
									AND (Pin1RETD AND Pin4RETD AND Pin8RETD)
									(*V16*)
									AND (Clamp5RETD AND Clamp38RETD AND Slide3RETD AND Slide5RETD AND Slide9RETD AND Slide12RETD AND Slide13RETD)
									(*V18*)
									AND (Pin3RETD AND Pin6RETD)
									(*V19*)
									AND (Pin2RETD AND Pin5RETD AND Pin7RETD);
		ELSE
			Unclamp_Step.1:= FALSE;

	END_IF									

									
	(*Third Stage Unclamping*)	(*V5, V10 RET, IF NOT Model 543, V7 RET*)
	IF (Model_ID<3) AND Repo_Reqs.0 THEN
					Unclamp_Step.2:= Unclamp_Step.1 AND TurntableA_At_Robot AND 
									(*V4*)
									(Clamp3RETD AND Clamp12RETD AND Clamp20RETD AND Clamp28RETD AND Clamp34RETD)
									(*V6*)
									AND (Clamp6RETD AND Clamp9RETD AND Clamp30RETD AND Clamp36RETD)
									(*V14*)
									AND (Slide1RETD AND Slide2RETD AND Slide14RETD AND Slide15RETD)
									(*V8*)
									AND (Clamp22RETD AND Clamp26RETD);
		ELSIF (Model_ID=3) AND Repo_Reqs.0 THEN
					Unclamp_Step.2:= Unclamp_Step.1 AND TurntableA_At_Robot AND
									(*V4*)
									(Clamp3RETD AND Clamp12RETD AND Clamp20RETD AND Clamp28RETD AND Clamp34RETD)
									(*V6*)
									AND (Clamp6RETD AND Clamp9RETD AND Clamp30RETD AND Clamp36RETD)
									(*V14*)
									AND (Slide1RETD AND Slide2RETD AND Slide14RETD AND Slide15RETD);
		ELSIF (Model_ID>3) AND Repo_Reqs.0 THEN
					Unclamp_Step.2:= Unclamp_Step.1 AND TurntableA_At_Robot AND
									(*V4*)
									(Clamp3RETD AND Clamp12RETD AND Clamp20RETD AND Clamp28RETD AND Clamp34RETD)
									(*V6*)
									AND (Clamp6RETD AND Clamp9RETD AND Clamp30RETD AND Clamp36RETD)
									(*V14*)
									AND (Slide1RETD AND Slide2RETD AND Slide14RETD AND Slide15RETD)
									(*V9*)
									AND (Clamp23RETD AND Clamp25RETD);
		ELSE
			Unclamp_Step.2:= FALSE;
	END_IF				
		
	(*Fourth Stage Unclamping*)	(*V1-V3, V12 RET, IF Model 543, V20, V21 RET*)
	IF NOT (Model_ID=3) AND (Unload_Complete AND TurntableB_At_Robot) (*AND All_Subs_Complete*) THEN
					Unclamp_Step.3:= (NOT Valve1FB.SideB_Indicator OR NOT Valve2FB.SideB_Indicator OR NOT Valve3FB.SideB_Indicator 
									OR NOT Valve12FB.SideB_Indicator) AND NOT Clamp_Step.0 AND 
									(*V5*)
									(Clamp4RETD AND Clamp11RETD AND Clamp21RETD AND Clamp29RETD AND Clamp33RETD)
									(*V10*)
									AND (Slide4RETD AND Slide8RETD AND Slide11RETD)
									(*V7*)
									AND (Clamp7RETD AND Clamp35RETD);
		ELSIF (Model_ID=3) AND (Unload_Complete) THEN
					Unclamp_Step.3:= TRUE;
		ELSE
			Unclamp_Step.3:= FALSE;					
	END_IF	
*)	

(*------------------------------------------- Repositions --------------------------------------*)

	(*Reposition Request#1*)
	IF (MAIN.R4.Peripheral_Req.0 AND (MAIN.R4.Task_ID_Ack=PickUp_Fix01))
		THEN
			Repo_Reqs.0:= TRUE;
	END_IF;

	(*Reposition Request#2*)
	IF FALSE
		THEN
			Repo_Reqs.1:= TRUE;
	END_IF;

	(*Reposition Request#3*)
	IF FALSE
		THEN
			Repo_Reqs.2:= TRUE;
	END_IF;

	(*Reposition Request#4*)
	IF FALSE
		THEN
			Repo_Reqs.3:= TRUE;
	END_IF;

	(*Reposition Request#5*)
	IF FALSE
		THEN
			Repo_Reqs.4:= TRUE;
	END_IF;

	(*Reposition Request#6*)
	IF FALSE
		THEN
			Repo_Reqs.5:= TRUE;
	END_IF;

	(*Reposition Request#7*)
	IF FALSE
		THEN
			Repo_Reqs.6:= TRUE;
	END_IF;

	(*Reposition Request#8*)
	IF FALSE
		THEN
			Repo_Reqs.7:= TRUE;
	END_IF;

	(*Reset All Reposition Acks At the End Of Cycle*)
	IF Cycle_Complete
		THEN
			Repo_Reqs:= 0;
	END_IF;

(*------------------------- Reposition Acks ---------------------*)
	Repo_Ack.0:= Repo_Reqs.0 AND Tool_At_Unload.1;
	Repo_Ack.1:= Repo_Reqs.1 AND FALSE;
	Repo_Ack.2:= Repo_Reqs.2 AND FALSE;
	Repo_Ack.3:= Repo_Reqs.3 AND FALSE;
	Repo_Ack.4:= Repo_Reqs.4 AND FALSE;
	Repo_Ack.5:= Repo_Reqs.5 AND FALSE;
	Repo_Ack.6:= Repo_Reqs.6 AND FALSE;
	Repo_Ack.7:= Repo_Reqs.7 AND FALSE;
END_ACTION

ACTION ValveBank1:


(*+++++++++++THIS AREA IS CUSTOM PER INSTALLATION AND WILL HAVE TO BE MODIFIED PER +++++++++++++*)
(*+++++++++++THIS AREA IS CUSTOM PER INSTALLATION AND WILL HAVE TO BE MODIFIED PER +++++++++++++*)
(*+++++++++++THIS AREA IS CUSTOM PER INSTALLATION AND WILL HAVE TO BE MODIFIED PER +++++++++++++*)

(*+++++++++++VALVE BANK 1 +++++++++++++*)
(*+++++++++++VALVE BANK 1 +++++++++++++*)
(*+++++++++++VALVE BANK 1 +++++++++++++*)


	(*Valve 1, A+B*)
	(*Clamps #1, 2, 32, 37*)
		Valve1FB
			(
			Enable_Motion:= Enable_Motion,
			Enable_Latch:= TRUE,					(*Enabling Runs Valve as detent type (maintained solenoids*)
			Enable_SideA_PreCharge:= FALSE,		(*Enabling Turns Side A PreCharge Active, reset when Side B is energized in Auto*)
			Enable_SideB_PreCharge:= FALSE,		(*Enabling Turns Side B PreCharge Active, reset when Side A is energized in Auto*)
			PreCharge_Time:= T#0.1S,
			Enable_Auto_Commands:= In_Auto,
			Enable_Manual_Commands:= In_Manual AND (All_Robots_Clear OR TurntableB_At_Robot),  (*TLK ADDED OR*)
			In_Manual_SideA_Command:= Discrete_In.ManReqs.0,
			In_Manual_SideB_Command:= (Discrete_In.ManReqs.1 OR Discrete_In.Go_Home),
			SideA_Indicator:= (Clamp1ADVD AND Clamp2ADVD AND Clamp32ADVD AND Clamp37ADVD),
			SideB_Indicator:= (Clamp1RETD AND Clamp2RETD AND Clamp32RETD AND Clamp37RETD) OR Manual_Ind_HomePrompt,
			TurnOn_SideA_SOL=> N100.Q.0,
			TurnOn_SideB_SOL=> N100.Q.1,
			TurnOn_SideA_Indicator=> Manual_Indicators1.0,
			TurnOn_SideB_Indicator=> Manual_Indicators1.1
			 );
		Valve1FB.In_Auto_SideA_Command:= Clamp_Step.2 AND NOT Unclamp_Step.3;
		Valve1FB.In_Auto_SideB_Command:= Unclamp_Step.3
										OR ((TurntableA_At_Robot OR Turntable_Bypassed) AND All_Sensors_Off AND Weld_Robots_Clear);


	(*Valve 2, A+B*)
	(*Clamps #13, 14, 15*)
		Valve2FB
			(
			Enable_Motion:= Enable_Motion,
			Enable_Latch:= TRUE,					(*Enabling Runs Valve as detent type (maintained solenoids*)
			Enable_SideA_PreCharge:= FALSE,		(*Enabling Turns Side A PreCharge Active, reset when Side B is energized in Auto*)
			Enable_SideB_PreCharge:= FALSE,		(*Enabling Turns Side B PreCharge Active, reset when Side A is energized in Auto*)
			PreCharge_Time:= T#0.10S,
			Enable_Auto_Commands:= In_Auto,
			Enable_Manual_Commands:= In_Manual AND (All_Robots_Clear OR TurntableB_At_Robot),  (*TLK ADDED OR*)
			In_Manual_SideA_Command:= Discrete_In.ManReqs.2,
			In_Manual_SideB_Command:= (Discrete_In.ManReqs.3 OR Discrete_In.Go_Home),
			SideA_Indicator:= Clamp13ADVD AND Clamp14ADVD AND Clamp15ADVD,
			SideB_Indicator:= (Clamp13RETD AND Clamp14RETD AND Clamp15RETD) OR Manual_Ind_HomePrompt,
			TurnOn_SideA_SOL=> N100.Q.2,
			TurnOn_SideB_SOL=> N100.Q.3,
			TurnOn_SideA_Indicator=> Manual_Indicators1.2,
			TurnOn_SideB_Indicator=> Manual_Indicators1.3
			 );
		Valve2FB.In_Auto_SideA_Command:= Clamp_Step.2 AND NOT Unclamp_Step.3;
		Valve2FB.In_Auto_SideB_Command:= Unclamp_Step.3
										OR ((TurntableA_At_Robot OR Turntable_Bypassed) AND All_Sensors_Off AND Weld_Robots_Clear);


	(*Valve 3, A+B*)
	(*Clamps #16-19*)
		Valve3FB
			(
			Enable_Motion:= Enable_Motion,
			Enable_Latch:= TRUE,					(*Enabling Runs Valve as detent type (maintained solenoids*)
			Enable_SideA_PreCharge:= FALSE,		(*Enabling Turns Side A PreCharge Active, reset when Side B is energized in Auto*)
			Enable_SideB_PreCharge:= FALSE,		(*Enabling Turns Side B PreCharge Active, reset when Side A is energized in Auto*)
			PreCharge_Time:= T#0.10S,
			Enable_Auto_Commands:= In_Auto,
			Enable_Manual_Commands:= In_Manual AND (All_Robots_Clear OR TurntableB_At_Robot),  (*TLK ADDED OR*)
			In_Manual_SideA_Command:= Discrete_In.ManReqs.4,
			In_Manual_SideB_Command:= (Discrete_In.ManReqs.5 OR Discrete_In.Go_Home),
			SideA_Indicator:= Clamp16ADVD AND Clamp17ADVD AND Clamp18ADVD AND Clamp19ADVD,
			SideB_Indicator:= (Clamp16RETD AND Clamp17RETD AND Clamp18RETD AND Clamp19RETD) OR Manual_Ind_HomePrompt,
			TurnOn_SideA_SOL=> N100.Q.4,
			TurnOn_SideB_SOL=> N100.Q.5,
			TurnOn_SideA_Indicator=> Manual_Indicators1.4,
			TurnOn_SideB_Indicator=> Manual_Indicators1.5
			 );
		Valve3FB.In_Auto_SideA_Command:= Clamp_Step.2 AND NOT Unclamp_Step.3;
		Valve3FB.In_Auto_SideB_Command:= Unclamp_Step.3
										OR ((TurntableA_At_Robot OR Turntable_Bypassed) AND All_Sensors_Off AND Weld_Robots_Clear);


	(*Valve 4, A+B*)
	(*Clamps #3, 12, 20, 28, 34*)
		Valve4FB
			(
			Enable_Motion:= Enable_Motion,
			Enable_Latch:= TRUE,					(*Enabling Runs Valve as detent type (maintained solenoids*)
			Enable_SideA_PreCharge:= FALSE,		(*Enabling Turns Side A PreCharge Active, reset when Side B is energized in Auto*)
			Enable_SideB_PreCharge:= FALSE,		(*Enabling Turns Side B PreCharge Active, reset when Side A is energized in Auto*)
			PreCharge_Time:= T#0.10S,
			Enable_Auto_Commands:= In_Auto,
			Enable_Manual_Commands:= In_Manual AND (All_Robots_Clear OR TurntableB_At_Robot),  (*TLK ADDED OR*)
			In_Manual_SideA_Command:= Discrete_In.ManReqs.6,
			In_Manual_SideB_Command:= (Discrete_In.ManReqs.7 OR Discrete_In.Go_Home),
			SideA_Indicator:= Clamp3ADVD AND Clamp12ADVD AND Clamp20ADVD AND Clamp28ADVD AND Clamp34ADVD,
			SideB_Indicator:= (Clamp3RETD AND Clamp12RETD AND Clamp20RETD AND Clamp28RETD AND Clamp34RETD) OR Manual_Ind_HomePrompt,
			TurnOn_SideA_SOL=> N100.Q.6,
			TurnOn_SideB_SOL=> N100.Q.7,
			TurnOn_SideA_Indicator=> Manual_Indicators1.6,
			TurnOn_SideB_Indicator=> Manual_Indicators1.7
			 );
		Valve4FB.In_Auto_SideA_Command:= Clamp_Step.2 AND NOT Unclamp_Step.1;
		Valve4FB.In_Auto_SideB_Command:= Unclamp_Step.1
										OR ((TurntableA_At_Robot OR Turntable_Bypassed) AND All_Sensors_Off AND Weld_Robots_Clear);


	(*Valve 5, A+B*)
	(*Clamps #4, 11, 21, 29, 33*) (*Added 21 TLK*)
		Valve5FB
			(
			Enable_Motion:= Enable_Motion,	
			Enable_Latch:= FALSE,					(*Enabling Runs Valve as detent type (maintained solenoids*)
			Enable_SideA_PreCharge:= FALSE,		(*Enabling Turns Side A PreCharge Active, reset when Side B is energized in Auto*)
			Enable_SideB_PreCharge:= FALSE,		(*Enabling Turns Side B PreCharge Active, reset when Side A is energized in Auto*)
			PreCharge_Time:= T#0.10S,
			Enable_Auto_Commands:= In_Auto,
			Enable_Manual_Commands:= In_Manual AND (All_Robots_Clear OR TurntableB_At_Robot),  (*TLK ADDED OR*)
			In_Manual_SideA_Command:= Discrete_In.ManReqs.8,
			In_Manual_SideB_Command:= (Discrete_In.ManReqs.9 OR Discrete_In.Go_Home),
			SideA_Indicator:= Clamp4ADVD AND Clamp11ADVD AND Clamp21ADVD AND Clamp29ADVD AND Clamp33ADVD, (*TLK ADDED Clamp21ADVD*)
			SideB_Indicator:= (Clamp4RETD AND Clamp11RETD AND Clamp21RETD AND Clamp29RETD AND Clamp33RETD) OR Manual_Ind_HomePrompt, (*TLK ADDED Clamp21RETD*)
			TurnOn_SideA_SOL=> N100.Q.8,
			TurnOn_SideB_SOL=> N100.Q.9,
			TurnOn_SideA_Indicator=> Manual_Indicators1.8,
			TurnOn_SideB_Indicator=> Manual_Indicators1.9
			 );
		Valve5FB.In_Auto_SideA_Command:= Clamp_Step.2 AND NOT Unclamp_Step.2;	
		Valve5FB.In_Auto_SideB_Command:= Unclamp_Step.2
										OR ((TurntableA_At_Robot OR Turntable_Bypassed) AND All_Sensors_Off AND Weld_Robots_Clear);


	(*Valve 6, A+B*)
	(*Clamps #6, 9, 30, 36*)
		Valve6FB
			(
			Enable_Motion:= Enable_Motion,
			Enable_Latch:= FALSE,					(*Enabling Runs Valve as detent type (maintained solenoids*)
			Enable_SideA_PreCharge:= FALSE,		(*Enabling Turns Side A PreCharge Active, reset when Side B is energized in Auto*)
			Enable_SideB_PreCharge:= FALSE,		(*Enabling Turns Side B PreCharge Active, reset when Side A is energized in Auto*)
			PreCharge_Time:= T#0.10S,
			Enable_Auto_Commands:= In_Auto,
			Enable_Manual_Commands:= In_Manual AND (All_Robots_Clear OR TurntableB_At_Robot),  (*TLK ADDED OR*)
			In_Manual_SideA_Command:= Discrete_In.ManReqs.10,
			In_Manual_SideB_Command:= (Discrete_In.ManReqs.11 OR Discrete_In.Go_Home),
			SideA_Indicator:= Clamp6ADVD AND Clamp9ADVD AND Clamp30ADVD AND Clamp36ADVD,
			SideB_Indicator:= (Clamp6RETD AND Clamp9RETD AND Clamp30RETD AND Clamp36RETD) OR Manual_Ind_HomePrompt,
			TurnOn_SideA_SOL=> N100.Q.10,
			TurnOn_SideB_SOL=> N100.Q.11,
			TurnOn_SideA_Indicator=> Manual_Indicators1.10,
			TurnOn_SideB_Indicator=> Manual_Indicators1.11
			 );
		Valve6FB.In_Auto_SideA_Command:= Clamp_Step.1 AND NOT Unclamp_Step.1;
		Valve6FB.In_Auto_SideB_Command:= Unclamp_Step.1
										OR ((TurntableA_At_Robot OR Turntable_Bypassed) AND All_Sensors_Off AND Weld_Robots_Clear);


	(*Valve 7, ALL BUT 543*)
	(*Clamps #7, 35*)
		Valve7FB
			(
			Enable_Motion:= Enable_Motion,
			Enable_Latch:= TRUE,					(*Enabling Runs Valve as detent type (maintained solenoids*)
			Enable_SideA_PreCharge:= FALSE,		(*Enabling Turns Side A PreCharge Active, reset when Side B is energized in Auto*)
			Enable_SideB_PreCharge:= FALSE,		(*Enabling Turns Side B PreCharge Active, reset when Side A is energized in Auto*)
			PreCharge_Time:= T#0.10S,
			Enable_Auto_Commands:= In_Auto,
			Enable_Manual_Commands:= In_Manual AND (All_Robots_Clear OR TurntableB_At_Robot),  (*TLK ADDED OR*)
			In_Manual_SideA_Command:= Discrete_In.ManReqs.12,
			In_Manual_SideB_Command:= (Discrete_In.ManReqs.13 OR Discrete_In.Go_Home),
			SideA_Indicator:= Clamp7ADVD AND Clamp35ADVD,
			SideB_Indicator:= (Clamp7RETD AND Clamp35RETD) OR Manual_Ind_HomePrompt,
			TurnOn_SideA_SOL=> N100.Q.12,
			TurnOn_SideB_SOL=> N100.Q.13,
			TurnOn_SideA_Indicator=> Manual_Indicators1.12,
			TurnOn_SideB_Indicator=> Manual_Indicators1.13
			 );
			 
	IF NOT ((Model_ID=3) OR (Model_ID=10)) THEN		 
				Valve7FB.In_Auto_SideA_Command:= Clamp_Step.2 AND NOT Unclamp_Step.2;
				Valve7FB.In_Auto_SideB_Command:= Unclamp_Step.2
												OR ((TurntableA_At_Robot OR Turntable_Bypassed) AND All_Sensors_Off AND Weld_Robots_Clear);
		ELSIF ((Model_ID=3) OR (Model_ID=10)) THEN
				Valve7FB.In_Auto_SideA_Command:= FALSE;
				Valve7FB.In_Auto_SideB_Command:= TRUE;
	END_IF
												
												

	(*Valve 8, ONLY 504, 524*)
	(*Clamps #22, 26*)
		Valve8FB
			(
			Enable_Motion:= Enable_Motion,
			Enable_Latch:= TRUE,					(*Enabling Runs Valve as detent type (maintained solenoids*)
			Enable_SideA_PreCharge:= FALSE,		(*Enabling Turns Side A PreCharge Active, reset when Side B is energized in Auto*)
			Enable_SideB_PreCharge:= FALSE,		(*Enabling Turns Side B PreCharge Active, reset when Side A is energized in Auto*)
			PreCharge_Time:= T#0.10S,
			Enable_Auto_Commands:= In_Auto,
			Enable_Manual_Commands:= In_Manual AND (All_Robots_Clear OR TurntableB_At_Robot),  (*TLK ADDED OR*)
			In_Manual_SideA_Command:= Discrete_In.ManReqs.14,
			In_Manual_SideB_Command:= (Discrete_In.ManReqs.15 OR Discrete_In.Go_Home),
			SideA_Indicator:= Clamp22ADVD AND Clamp26ADVD,
			SideB_Indicator:= (Clamp22RETD AND Clamp26RETD) OR Manual_Ind_HomePrompt,
			TurnOn_SideA_SOL=> N100.Q.14,
			TurnOn_SideB_SOL=> N100.Q.15,
			TurnOn_SideA_Indicator=> Manual_Indicators1.14,
			TurnOn_SideB_Indicator=> Manual_Indicators1.15
			 );
			 
	IF (*(Model_ID<3)*) (Model_ID=1) OR (Model_ID=2) OR (Model_ID=8) OR (Model_ID=9) THEN		 
				Valve8FB.In_Auto_SideA_Command:= (Clamp_Step.2 AND NOT Unclamp_Step.1);
				Valve8FB.In_Auto_SideB_Command:= Unclamp_Step.1
												OR ((TurntableA_At_Robot OR Turntable_Bypassed) AND All_Sensors_Off AND Weld_Robots_Clear);
		ELSE
				Valve8FB.In_Auto_SideA_Command:= FALSE;
				Valve8FB.In_Auto_SideB_Command:= TRUE;
		END_IF

	(*Valve 9, ONLY 526, 536, 550, 571*)
	(*Clamp #23, 25*)
		Valve9FB
			(
			Enable_Motion:= Enable_Motion,
			Enable_Latch:= TRUE,					(*Enabling Runs Valve as detent type (maintained solenoids*)
			Enable_SideA_PreCharge:= FALSE,		(*Enabling Turns Side A PreCharge Active, reset when Side B is energized in Auto*)
			Enable_SideB_PreCharge:= FALSE,		(*Enabling Turns Side B PreCharge Active, reset when Side A is energized in Auto*)
			PreCharge_Time:= T#0.10S,
			Enable_Auto_Commands:= In_Auto,
			Enable_Manual_Commands:= In_Manual AND (All_Robots_Clear OR TurntableB_At_Robot),  (*TLK ADDED OR*)
			In_Manual_SideA_Command:= Discrete_In.ManReqs.16,
			In_Manual_SideB_Command:= (Discrete_In.ManReqs.17 OR Discrete_In.Go_Home),
			SideA_Indicator:= Clamp23ADVD AND Clamp25ADVD,
			SideB_Indicator:= (Clamp23RETD AND Clamp25RETD) OR Manual_Ind_HomePrompt,
			TurnOn_SideA_SOL=> N100.Q.16,
			TurnOn_SideB_SOL=> N100.Q.17,
			TurnOn_SideA_Indicator=> Manual_Indicators1.16,
			TurnOn_SideB_Indicator=> Manual_Indicators1.17
			 );
			 
	IF (*(Model_ID>3)*)    (Model_ID=4) OR (Model_ID=5) OR (Model_ID=6) OR (Model_ID=7)
						OR (Model_ID=11) OR (Model_ID=12) OR (Model_ID=13) OR (Model_ID=14)
						OR (Model_ID=15) OR (Model_ID=16) OR (Model_ID=17) OR (Model_ID=18)
						OR (Model_ID=19) OR (Model_ID=20) OR (Model_ID=21) OR (Model_ID=22)  THEN		 
				Valve9FB.In_Auto_SideA_Command:= (Clamp_Step.2 AND NOT Unclamp_Step.1);
				Valve9FB.In_Auto_SideB_Command:= Unclamp_Step.1
												OR ((TurntableA_At_Robot OR Turntable_Bypassed) AND All_Sensors_Off AND Weld_Robots_Clear);
		ELSE
				Valve9FB.In_Auto_SideA_Command:= FALSE;
				Valve9FB.In_Auto_SideB_Command:= TRUE;
		END_IF

	(*Valve 10, A+B*)
	(*Slides #4, 8, 11*)
		Valve10FB
			(
			Enable_Motion:= Enable_Motion,
			Enable_Latch:= TRUE,					(*Enabling Runs Valve as detent type (maintained solenoids*)
			Enable_SideA_PreCharge:= FALSE,		(*Enabling Turns Side A PreCharge Active, reset when Side B is energized in Auto*)
			Enable_SideB_PreCharge:= FALSE,		(*Enabling Turns Side B PreCharge Active, reset when Side A is energized in Auto*)
			PreCharge_Time:= T#0.10S,
			Enable_Auto_Commands:= In_Auto,
			Enable_Manual_Commands:= In_Manual AND (All_Robots_Clear OR TurntableB_At_Robot),  (*TLK ADDED OR*)
			In_Manual_SideA_Command:= (Discrete_In.ManReqs.18 OR Discrete_In.Go_Home),
			In_Manual_SideB_Command:= Discrete_In.ManReqs.19,
			SideA_Indicator:= (Slide4ADVD AND Slide8ADVD AND Slide11ADVD) OR Manual_Ind_HomePrompt,
			SideB_Indicator:= Slide4RETD AND Slide8RETD AND Slide11RETD,
			TurnOn_SideA_SOL=> N100.Q.18,
			TurnOn_SideB_SOL=> N100.Q.19,
			TurnOn_SideA_Indicator=> Manual_Indicators1.18,
			TurnOn_SideB_Indicator=> Manual_Indicators1.19
			 );
		Valve10FB.In_Auto_SideA_Command:= (Clamp_Step.0 AND NOT Unclamp_Step.2 OR Unclamp_Step.3)
										OR ((TurntableA_At_Robot OR Turntable_Bypassed) AND All_Sensors_Off AND Weld_Robots_Clear);
		Valve10FB.In_Auto_SideB_Command:= Unclamp_Step.2;


	(*Valve 11, A+B*)
	(*Slide #6*)
		Valve11FB
			(
			Enable_Motion:= Enable_Motion,
			Enable_Latch:= TRUE,					(*Enabling Runs Valve as detent type (maintained solenoids*)
			Enable_SideA_PreCharge:= FALSE,		(*Enabling Turns Side A PreCharge Active, reset when Side B is energized in Auto*)
			Enable_SideB_PreCharge:= FALSE,		(*Enabling Turns Side B PreCharge Active, reset when Side A is energized in Auto*)
			PreCharge_Time:= T#0.10S,
			Enable_Auto_Commands:= In_Auto,
			Enable_Manual_Commands:= In_Manual AND (All_Robots_Clear OR TurntableB_At_Robot),  (*TLK ADDED OR*)
			In_Manual_SideA_Command:= (Discrete_In.ManReqs.20 OR Discrete_In.Go_Home),
			In_Manual_SideB_Command:= Discrete_In.ManReqs.21,
			SideA_Indicator:= (Slide6ADVD) OR Manual_Ind_HomePrompt,
			SideB_Indicator:= Slide6RETD,
			TurnOn_SideA_SOL=> N100.Q.20,
			TurnOn_SideB_SOL=> N100.Q.21,
			TurnOn_SideA_Indicator=> Manual_Indicators1.20,
			TurnOn_SideB_Indicator=> Manual_Indicators1.21
			 );
		Valve11FB.In_Auto_SideA_Command:= (Clamp_Step.0 AND NOT Unclamp_Step.0 OR Unclamp_Step.3)
										OR ((TurntableA_At_Robot OR Turntable_Bypassed) AND All_Sensors_Off AND Weld_Robots_Clear);
		Valve11FB.In_Auto_SideB_Command:= Unclamp_Step.0;


	(*Valve 12, A+B*)
	(*Slide #7*)
		Valve12FB
			(
			Enable_Motion:= Enable_Motion,
			Enable_Latch:= TRUE,					(*Enabling Runs Valve as detent type (maintained solenoids*)
			Enable_SideA_PreCharge:= FALSE,		(*Enabling Turns Side A PreCharge Active, reset when Side B is energized in Auto*)
			Enable_SideB_PreCharge:= FALSE,		(*Enabling Turns Side B PreCharge Active, reset when Side A is energized in Auto*)
			PreCharge_Time:= T#0.10S,
			Enable_Auto_Commands:= In_Auto,
			Enable_Manual_Commands:= In_Manual AND (All_Robots_Clear OR TurntableB_At_Robot),  (*TLK ADDED OR*)
			In_Manual_SideA_Command:= Discrete_In.ManReqs.22,
			In_Manual_SideB_Command:= (Discrete_In.ManReqs.23 OR Discrete_In.Go_Home),
			SideA_Indicator:= Slide7ADVD,
			SideB_Indicator:= (Slide7RETD) OR Manual_Ind_HomePrompt,
			TurnOn_SideA_SOL=> N100.Q.22,
			TurnOn_SideB_SOL=> N100.Q.23,
			TurnOn_SideA_Indicator=> Manual_Indicators1.22,
			TurnOn_SideB_Indicator=> Manual_Indicators1.23
			 );
		Valve12FB.In_Auto_SideA_Command:= Clamp_Step.1 AND NOT Unclamp_Step.3;
		Valve12FB.In_Auto_SideB_Command:= Unclamp_Step.3
										OR ((TurntableA_At_Robot OR Turntable_Bypassed) AND All_Sensors_Off AND Weld_Robots_Clear);


	(*Valve 13, A+B*)
	(*Slide #10*)
		Valve13FB
			(
			Enable_Motion:= Enable_Motion,
			Enable_Latch:= FALSE,					(*Enabling Runs Valve as detent type (maintained solenoids*)
			Enable_SideA_PreCharge:= FALSE,		(*Enabling Turns Side A PreCharge Active, reset when Side B is energized in Auto*)
			Enable_SideB_PreCharge:= FALSE,		(*Enabling Turns Side B PreCharge Active, reset when Side A is energized in Auto*)
			PreCharge_Time:= T#0.10S,
			Enable_Auto_Commands:= In_Auto,
			Enable_Manual_Commands:= In_Manual AND (All_Robots_Clear OR TurntableB_At_Robot),  (*TLK ADDED OR*)
			In_Manual_SideA_Command:= Discrete_In.ManReqs.24,
			In_Manual_SideB_Command:= (Discrete_In.ManReqs.25 OR Discrete_In.Go_Home),
			SideA_Indicator:= Slide10ADVD,
			SideB_Indicator:= (Slide10RETD) OR Manual_Ind_HomePrompt,
			TurnOn_SideA_SOL=> N100.Q.24,
			TurnOn_SideB_SOL=> N100.Q.25,
			TurnOn_SideA_Indicator=> Manual_Indicators1.24,
			TurnOn_SideB_Indicator=> Manual_Indicators1.25
			 );
		IF (*(Model_ID>3)*)    	   (Model_ID=4) OR (Model_ID=5) OR (Model_ID=6) OR (Model_ID=7)
								OR (Model_ID=11) OR (Model_ID=12) OR (Model_ID=13) OR (Model_ID=14)
								OR (Model_ID=15) OR (Model_ID=16) OR (Model_ID=17) OR (Model_ID=18)
								OR (Model_ID=19) OR (Model_ID=20) OR (Model_ID=21) OR (Model_ID=22) THEN	
		Valve13FB.In_Auto_SideA_Command:= (Clamp_Step.1 AND NOT Unclamp_Step.0);
		Valve13FB.In_Auto_SideB_Command:= Unclamp_Step.0
										OR ((TurntableA_At_Robot OR Turntable_Bypassed) AND All_Sensors_Off AND Weld_Robots_Clear);
		ELSE
		Valve13FB.In_Auto_SideB_Command:=TRUE;
		END_IF


	(*Valve 14, A+B*)
	(*Slide #1, 2, 14, 15*)
		Valve14FB
			(
			Enable_Motion:= Enable_Motion,
			Enable_Latch:= TRUE,					(*Enabling Runs Valve as detent type (maintained solenoids*)
			Enable_SideA_PreCharge:= FALSE,		(*Enabling Turns Side A PreCharge Active, reset when Side B is energized in Auto*)
			Enable_SideB_PreCharge:= FALSE,		(*Enabling Turns Side B PreCharge Active, reset when Side A is energized in Auto*)
			PreCharge_Time:= T#0.10S,
			Enable_Auto_Commands:= In_Auto,
			Enable_Manual_Commands:= In_Manual AND (All_Robots_Clear OR TurntableB_At_Robot),  (*TLK ADDED OR*)
			In_Manual_SideA_Command:= (Discrete_In.ManReqs.26 OR Discrete_In.Go_Home),
			In_Manual_SideB_Command:=  Discrete_In.ManReqs.27,
			SideA_Indicator:= (Slide1ADVD AND Slide2ADVD AND Slide14ADVD AND Slide15ADVD) OR Manual_Ind_HomePrompt,
			SideB_Indicator:=  Slide1RETD AND Slide2RETD AND Slide14RETD AND Slide15RETD,
			TurnOn_SideA_SOL=> N100.Q.26,
			TurnOn_SideB_SOL=> N100.Q.27,
			TurnOn_SideA_Indicator=> Manual_Indicators1.26,
			TurnOn_SideB_Indicator=> Manual_Indicators1.27
			 );
		Valve14FB.In_Auto_SideA_Command:= (Clamp_Step.0 AND NOT Unclamp_Step.1 OR Unclamp_Step.3)
										OR ((TurntableA_At_Robot OR Turntable_Bypassed) AND All_Sensors_Off AND Weld_Robots_Clear);
		Valve14FB.In_Auto_SideB_Command:= Unclamp_Step.1;


	(*Valve 15, A+B*)
	(*Pin #1, 4, 8*)
		Valve15FB
			(
			Enable_Motion:= Enable_Motion,
			Enable_Latch:= TRUE,					(*Enabling Runs Valve as detent type (maintained solenoids*)
			Enable_SideA_PreCharge:= FALSE,		(*Enabling Turns Side A PreCharge Active, reset when Side B is energized in Auto*)
			Enable_SideB_PreCharge:= FALSE,		(*Enabling Turns Side B PreCharge Active, reset when Side A is energized in Auto*)
			PreCharge_Time:= T#0.10S,
			Enable_Auto_Commands:= In_Auto,
			Enable_Manual_Commands:= In_Manual AND (All_Robots_Clear OR TurntableB_At_Robot),  (*TLK ADDED OR*)
			In_Manual_SideA_Command:= (Discrete_In.ManReqs.28 OR Discrete_In.Go_Home),
			In_Manual_SideB_Command:= Discrete_In.ManReqs.29,
			SideA_Indicator:= (Pin1ADVD AND Pin4ADVD AND Pin8ADVD) OR Manual_Ind_HomePrompt,
			SideB_Indicator:= Pin1RETD AND Pin4RETD AND Pin8RETD,
			TurnOn_SideA_SOL=> N100.Q.28,
			TurnOn_SideB_SOL=> N100.Q.29,
			TurnOn_SideA_Indicator=> Manual_Indicators1.28,
			TurnOn_SideB_Indicator=> Manual_Indicators1.29
			 );
		Valve15FB.In_Auto_SideA_Command:= (Clamp_Step.0 AND NOT Unclamp_Step.0 OR Unclamp_Step.3)
										OR ((TurntableA_At_Robot OR Turntable_Bypassed) AND All_Sensors_Off AND Weld_Robots_Clear);
		Valve15FB.In_Auto_SideB_Command:= Unclamp_Step.0;


	(*Valve 16, A+B*)
	(*Clamp #5, 38, Slide #3, 5, 9, 12, 13*)
		Valve16FB
			(
			Enable_Motion:= Enable_Motion,
			Enable_Latch:= TRUE,					(*Enabling Runs Valve as detent type (maintained solenoids*)
			Enable_SideA_PreCharge:= FALSE,		(*Enabling Turns Side A PreCharge Active, reset when Side B is energized in Auto*)
			Enable_SideB_PreCharge:= FALSE,		(*Enabling Turns Side B PreCharge Active, reset when Side A is energized in Auto*)
			PreCharge_Time:= T#0.10S,
			Enable_Auto_Commands:= In_Auto,
			Enable_Manual_Commands:= In_Manual AND (All_Robots_Clear OR TurntableB_At_Robot),  (*TLK ADDED OR*)
			In_Manual_SideA_Command:= Discrete_In.ManReqs.30,
			In_Manual_SideB_Command:= (Discrete_In.ManReqs.31 OR Discrete_In.Go_Home),
			SideA_Indicator:= Clamp5ADVD AND Clamp38ADVD AND Slide3ADVD AND Slide5ADVD AND Slide9ADVD AND Slide12ADVD AND Slide13ADVD,
			SideB_Indicator:= (Clamp5RETD AND Clamp38RETD AND Slide3RETD AND Slide5RETD AND Slide9RETD AND Slide12RETD AND Slide13RETD) OR Manual_Ind_HomePrompt,
			TurnOn_SideA_SOL=> N100.Q.30,
			TurnOn_SideB_SOL=> N100.Q.31,
			TurnOn_SideA_Indicator=> Manual_Indicators1.30,
			TurnOn_SideB_Indicator=> Manual_Indicators1.31
			 );
		Valve16FB.In_Auto_SideA_Command:= (Clamp_Step.4 AND NOT Unclamp_Step.0);
		Valve16FB.In_Auto_SideB_Command:= Unclamp_Step.0
										OR ((TurntableA_At_Robot OR Turntable_Bypassed) AND All_Sensors_Off AND Weld_Robots_Clear);


























(*end*)
END_ACTION

ACTION ValveBank2:


(*+++++++++++THIS AREA IS CUSTOM PER INSTALLATION AND WILL HAVE TO BE MODIFIED PER +++++++++++++*)
(*+++++++++++THIS AREA IS CUSTOM PER INSTALLATION AND WILL HAVE TO BE MODIFIED PER +++++++++++++*)
(*+++++++++++THIS AREA IS CUSTOM PER INSTALLATION AND WILL HAVE TO BE MODIFIED PER +++++++++++++*)

(*+++++++++++VALVE BANK 2 +++++++++++++*)
(*+++++++++++VALVE BANK 2 +++++++++++++*)
(*+++++++++++VALVE BANK 2 +++++++++++++*)


	(*Valve 17, A+B*)
	(*QA Checks #1-6*)
		Valve17FB
			(
			Enable_Motion:= Enable_Motion ,
			Enable_Latch:= TRUE,					(*Enabling Runs Valve as detent type (maintained solenoids*)
			Enable_SideA_PreCharge:= FALSE,		(*Enabling Turns Side A PreCharge Active, reset when Side B is energized in Auto*)
			Enable_SideB_PreCharge:= FALSE,		(*Enabling Turns Side B PreCharge Active, reset when Side A is energized in Auto*)
			PreCharge_Time:= T#0.1S,
			Enable_Auto_Commands:= In_Auto,
			Enable_Manual_Commands:= In_Manual AND (All_Robots_Clear OR TurntableB_At_Robot),  (*TLK ADDED OR*)
			In_Manual_SideA_Command:= Discrete_In.ManReqs2.0,
			In_Manual_SideB_Command:= (Discrete_In.ManReqs2.1 OR Discrete_In.Go_Home),
			SideA_Indicator:= QACheck1ADVD AND QACheck2ADVD AND QACheck3ADVD AND QACheck4ADVD AND QACheck5ADVD AND QACheck6ADVD,
			SideB_Indicator:= (QACheck1RETD AND QACheck2RETD AND QACheck3RETD AND QACheck4RETD AND QACheck5RETD AND QACheck6RETD) OR Manual_Ind_HomePrompt,
			TurnOn_SideA_SOL=> N101.Q.0,
			TurnOn_SideB_SOL=> N101.Q.1,
			TurnOn_SideA_Indicator=> Manual_Indicators2.0,
			TurnOn_SideB_Indicator=> Manual_Indicators2.1
			 );
		Valve17FB.In_Auto_SideA_Command:= CheckQA1FB.Fire_QAchecks AND NOT Cycle_Complete;
		Valve17FB.In_Auto_SideB_Command:= NOT CheckQA1FB.Fire_QAchecks OR (Cycle_Complete AND All_Sensors_Off);


